(* ======================================Schrittkette======================================== *)
fb_state_entry(
	i16_next_step:= ,
	i16_pos:= 1,
	s_debugtext:= ,
	E=> ,
	X=> ,
	i16_step=> ,
	i16_last_step=> );

CASE fb_state_entry.i16_step OF
(*=======================================================*)
	INIT_OBJ:
		IF st_config_achse.b_config_fertig THEN
			fb_state_entry.i16_next_step := 2;
		END_IF

(*=======================================================*)
	2:	(* Antriebsbegrenzende Konstantwerte *)
		IF fb_state_entry.E THEN
			CASE gst_datensatz.st_md.i16_typ_zelle OF
				KEINE_ZELLE:
					;

				BESTUECKZELLE_1700 :
					st_geschwindigkeiten.lr_auto_max := 350;	(* Hub/min *)
					st_geschwindigkeiten.lr_auto_min := 15;
					st_geschwindigkeiten.lr_jog := 50;
					gst_datensatz.st_md.st_md_bestueckachse.lr_startposition := 17;

				BESTUECKZELLE_1720:
					st_geschwindigkeiten.lr_auto_max := 300;	(* Hub/min *)
					st_geschwindigkeiten.lr_auto_min := 15;
					st_geschwindigkeiten.lr_jog := 50;
					gst_datensatz.st_md.st_md_bestueckachse.lr_startposition := 3;

				RASTERFOLIE:
					st_geschwindigkeiten.lr_auto_max := 300;	(* Hub/min *)
					st_geschwindigkeiten.lr_auto_min := 15;
					st_geschwindigkeiten.lr_jog := 50;
					gst_datensatz.st_md.st_md_bestueckachse.lr_startposition := 17;
			END_CASE

			fb_state_entry.i16_next_step := 3;
		END_IF

(*=======================================================*)
	3:	(* Spezifische NC-Achsparameter auslesen *)
		IF fb_state_entry.E THEN
			subr_ST_Bandeinzugsnocken_ein();
			fb_virt_master_axis.i16_nc_parameter_nummer := MaxVelocitySystem;
			st_drive_cmd.enu_cmd := READ_NC_PARAMETER;
		END_IF

		(*-----------------------Weiterschaltbedingungen----------------------------*)
		IF st_drive_cmd.enu_cmd = NO_COMMAND THEN
			st_geschwindigkeiten.lr_maximalgeschwindigkeit := fb_virt_master_axis.r_wert_nc_read_parameter(* °/s *) * 60 / 360;
			fb_state_entry.i16_next_step := 4;
		END_IF

(*=======================================================*)
	4:	(* Spezifische NC-Achsparameter auslesen *)
		IF fb_state_entry.E THEN
			fb_virt_master_axis.i16_nc_parameter_nummer := MaxAccelerationSystem;
			st_drive_cmd.enu_cmd := READ_NC_PARAMETER;
		END_IF

		(*-----------------------Weiterschaltbedingungen----------------------------*)
		IF st_drive_cmd.enu_cmd = NO_COMMAND THEN
			st_geschwindigkeiten.lr_beschleunigung := fb_virt_master_axis.r_wert_nc_read_parameter;
			fb_state_entry.i16_next_step := 5;
		END_IF

(*=======================================================*)
	5:	(* Spezifische NC-Achsparameter auslesen *)
		IF fb_state_entry.E THEN
			fb_virt_master_axis.i16_nc_parameter_nummer := MaxDecelerationSystem;
			st_drive_cmd.enu_cmd := READ_NC_PARAMETER;
		END_IF

		(*-----------------------Weiterschaltbedingungen----------------------------*)
		IF st_drive_cmd.enu_cmd = NO_COMMAND THEN
			st_geschwindigkeiten.lr_verzoegerung := fb_virt_master_axis.r_wert_nc_read_parameter;
			lr_decceleration_normal := st_geschwindigkeiten.lr_verzoegerung;
			lr_decceleration_nothalt := 200000.0;
			fb_state_entry.i16_next_step := 6;
		END_IF

(*=======================================================*)
	6:	(* Spezifische NC-Achsparameter auslesen *)
		IF fb_state_entry.E THEN
			fb_virt_master_axis.i16_nc_parameter_nummer := MaxJerk;
			st_drive_cmd.enu_cmd := READ_NC_PARAMETER;
		END_IF

		(*-----------------------Weiterschaltbedingungen----------------------------*)
		IF st_drive_cmd.enu_cmd = NO_COMMAND THEN
			st_geschwindigkeiten.lr_ruck := fb_virt_master_axis.r_wert_nc_read_parameter;
		fb_state_entry.i16_next_step := FEHLER; (*in Fehler gehen damit die Achsen resetet werden. Sonst steigen die Achsen bei einem TC Restart aus*)
		END_IF

(*=======================================================*)
	INIT:
		IF fb_state_entry.E THEN
			fb_ton_wz.IN := FALSE;
			fb_ton_uez.IN	:= FALSE;
			fb_ton_quitt.IN := FALSE;
			fb_ton_wz_disable.IN := FALSE;
			st_ctrl_out.b_fehler := FALSE;
			st_ctrl_out.b_fertig := FALSE;
			st_ctrl_out.b_bereit := FALSE;
			st_ctrl_out.b_prebereit := FALSE;
			b_merker_bandende_links := FALSE;
			b_merker_bandende_rechts := FALSE;

			(* Reset Stoermeldungen *)
			st_sm.b_achse_nicht_auf_startpos := FALSE;
			st_sm.b_achsfehler := FALSE;
			st_sm.b_devicefehler := FALSE;
			st_sm.b_keine_verfahrfreigabe := FALSE;
			st_sm.b_ende_skalierungs_nocke := FALSE;
			st_sm.b_ende_camming_nocke := FALSE;
			st_sm.b_skalierung_noch_aktiv := FALSE;
			sm_fehler_bestueckanzahl := FALSE;
			sm_fehler_bestueckposition_z := FALSE;
			sm_fehler_positionierung_z := FALSE;
			sm_fehler_bestueckposition_y := FALSE;
			sm_fehler_positionierung_y := FALSE;
			sm_fehler_achse_lueften := FALSE;
			sm_fehler_raster_oder_zaehne := FALSE;
			sm_fehler_bestueckschieberanzahl := FALSE;
			sm_keine_busverbindung := FALSE;
			sm_fehler_nach_bandwechsel := FALSE;
			sm_fehler_positionierung_bestueckachse := FALSE;

			(* Reset Betriebsmeldungen *)
			bm_bandende_einzug_links_erreicht := FALSE;
			bm_bandende_einzug_rechts_erreicht := FALSE;
			bm_bandende_beide_einzuege_erreicht := FALSE;
			bm_einzug_links_band_entnehmen := FALSE;
			bm_einzug_links_band_auf_anschlag := FALSE;
			bm_einzug_rechts_band_entnehmen := FALSE;
			bm_einzug_rechts_band_auf_anschlag := FALSE;
			bm_einzug_rechts_band_bis_gls := FALSE;
			bm_einzug_links_band_bis_gls := FALSE;
			bm_beide_Bandklemmen_oeffnen := FALSE;
			bm_an_visu_hinten := '';

			ST_TippTasten.b_einfaedeln_aktiv := FALSE;
			bandwechsel_kontroller.st_ctrl.in.b_start := FALSE;
			einpresskraft_kontroller.st_ctrl.in.b_start := FALSE;
			bandeinzug_kontroller.st_ctrl.in.b_freigabe := FALSE;
			axis_bandeinzug_achse.st_ctrl.in.b_freigabe := FALSE;
			axis_bandeinzug_achse.st_ctrl.in.b_bremse_auf := FALSE;
			axis_bandeinzug_achse.st_ctrl.in.b_bremse_zu := FALSE;
			axis_bandeinzug_achse.st_ctrl.in.b_start_schreiben := FALSE;
			axis_bandeinzug_achse.st_ctrl.in.b_start := FALSE;
			axis_bandeinzug_achse.st_ctrl.in.b_home := FALSE;
			axis_bandeinzug_achse.st_ctrl.in.b_ausfaedeln_servo := FALSE;
			axis_bandeinzug_achse.st_ctrl.in.b_einfaedeln_servo := FALSE;

			fb_berechnung_override_achse.lr_skalierung_slave_achse1 := 1;
			fb_berechnung_override_achse.lr_skalierung_slave_achse2 := 1;

			i16_step_lueften := 0;
			i16_einfaedelzaehler := 0;

			st_geschwindigkeiten.lr_verzoegerung := lr_decceleration_normal;

			b_bestueckschieber_ueberwachung_aktiv := TRUE;

			b_einfaedeln_aktiv_servo := FALSE;

			gb_memEndOfBandMarkNIO := FALSE;
		END_IF

		(* Gearout/Camout der Slaveachsen, damit diese quittiert werden können *)
		CASE gst_datensatz.st_md.i16_typ_zelle OF
			KEINE_ZELLE:
				;

			BESTUECKZELLE_1700:
				IF bestueckachse.NcToPlc.CoupleState > 0 THEN
					st_drive_cmd_bestueckachse.enu_cmd := CAM_OUT_SLAVE;
				END_IF
				IF z_achse.NcToPlc.CoupleState > 0 THEN
					st_drive_cmd_z_achse.enu_cmd := CAM_OUT_SLAVE;
				END_IF
				IF y_achse.NcToPlc.CoupleState > 0 THEN
					st_drive_cmd_y_achse.enu_cmd := CAM_OUT_SLAVE;
				END_IF

				CASE gst_datensatz.st_wkz.i16_typ_bandeinzug OF
					KEIN_EINZUG:
						;
					STANDARD_2FACH_V2:
						;
					 BANDWECHSLER_V2:
						;
					SERVO:
						IF b_achse.NcToPlc.CoupleState > 0 THEN
							st_drive_cmd_b_achse.enu_cmd := CAM_OUT_SLAVE;
						END_IF
				END_CASE

			BESTUECKZELLE_1720:
				IF bestueckachse.NcToPlc.CoupleState > 0 THEN
					st_drive_cmd_bestueckachse.enu_cmd := CAM_OUT_SLAVE;
				END_IF
				IF z_achse.NcToPlc.CoupleState > 0 THEN
					st_drive_cmd_z_achse.enu_cmd := CAM_OUT_SLAVE;
				END_IF

			RASTERFOLIE:
				IF bestueckachse.NcToPlc.CoupleState > 0 THEN
					st_drive_cmd_bestueckachse.enu_cmd := CAM_OUT_SLAVE;
				END_IF
				IF z_achse.NcToPlc.CoupleState > 0 THEN
					st_drive_cmd_z_achse.enu_cmd := CAM_OUT_SLAVE;
				END_IF
		END_CASE

		(*-----------------------Weiterschaltbedingungen----------------------------*)
		IF st_ctrl_in.b_preinit THEN
			fb_state_entry.i16_next_step := 12;
		END_IF

(*=======================================================*)
	12:	(* Reglerfreigabe wegnehmen *)
		IF fb_state_entry.E THEN
			st_drive_cmd.enu_cmd := POWER_DISABLE;
		END_IF

		(*-----------------------Weiterschaltbedingungen----------------------------*)
		IF st_drive_cmd.enu_cmd = NO_COMMAND THEN
			fb_state_entry.i16_next_step := 14;
		END_IF

(*=======================================================*)
	14:	(* Lade Wkz von Festplatte *)
		IF fb_state_entry.E THEN
			gi16_bbgen_auftrag := LESE_WKZ;
		END_IF

		IF  gi16_bbgen_auftrag = KEIN_BB_AUFTRAG THEN
			fb_ton_wz.pt := t#5ms;
			fb_ton_wz.IN := TRUE;
		END_IF

		IF fb_ton_wz.Q THEN
			fb_state_entry.i16_next_step := 16;
			fb_ton_wz.IN := FALSE;
		END_IF

(*=======================================================*)
	16: (* Band aus DB von Festplatte einlesen. *)
		IF fb_state_entry.E THEN
			gi16_bbgen_auftrag := LESE_BAND;
		END_IF

		IF  gi16_bbgen_auftrag = KEIN_BB_AUFTRAG THEN
			fb_ton_wz.pt := t#5ms;
			fb_ton_wz.IN := TRUE;
		END_IF

		IF fb_ton_wz.Q THEN
			fb_state_entry.i16_next_step := 20;
			fb_ton_wz.IN := FALSE;
		END_IF

(*=======================================================*)
	20:	(* CAM_OUT Bestückachse *)
		IF fb_state_entry.E THEN
			st_drive_cmd_bestueckachse.enu_cmd := CAM_OUT_SLAVE;
		END_IF

		(*-----------------------Weiterschaltbedingungen----------------------------*)
		IF st_drive_cmd_bestueckachse.enu_cmd = NO_COMMAND AND NOT fb_state_entry.E THEN
			fb_state_entry.i16_next_step := 30;
		END_IF

(*=======================================================*)
	30:	(* CAM Out Z-Achse *)
		IF fb_state_entry.E THEN
			st_drive_cmd_z_achse.enu_cmd := CAM_OUT_SLAVE;
		END_IF

		(*-----------------------Weiterschaltbedingungen----------------------------*)
		IF st_drive_cmd_z_achse.enu_cmd = NO_COMMAND AND NOT fb_state_entry.E THEN
			CASE gst_datensatz.st_md.i16_typ_zelle OF
				KEINE_ZELLE:
					;

				BESTUECKZELLE_1700:
					CASE gst_datensatz.st_wkz.i16_typ_bandeinzug OF
						KEIN_EINZUG,  STANDARD_2FACH_V2,  BANDWECHSLER_V2:
							fb_state_entry.i16_next_step := 40;
						SERVO:
							fb_state_entry.i16_next_step := 35;
					END_CASE;

				RASTERFOLIE:
					fb_state_entry.i16_next_step := 40;

				BESTUECKZELLE_1720:
					fb_state_entry.i16_next_step := 45;
			END_CASE
		END_IF

(*=======================================================*)
	35:	(* CAM Out B-Achse *)
		IF fb_state_entry.E THEN
			st_drive_cmd_b_achse.enu_cmd := CAM_OUT_SLAVE;
		END_IF

		(*-----------------------Weiterschaltbedingungen----------------------------*)
		IF st_drive_cmd_b_achse.enu_cmd = NO_COMMAND AND NOT fb_state_entry.E THEN
			fb_state_entry.i16_next_step := 40;
		END_IF

(*=======================================================*)
	40:	(* CAM Out Y-Achse *)
		IF fb_state_entry.E THEN
			st_drive_cmd_y_achse.enu_cmd := CAM_OUT_SLAVE;
		END_IF

		(*-----------------------Weiterschaltbedingungen----------------------------*)
		IF st_drive_cmd_y_achse.enu_cmd = NO_COMMAND AND NOT fb_state_entry.E THEN
			fb_state_entry.i16_next_step := 45;
		END_IF

(*=======================================================*)
	45:	(* Reglerfreigabe setzen , Reset wird bei Bedarf automatisch ausgeführt*)
		IF fb_state_entry.E THEN
			st_drive_cmd.enu_cmd := POWER_ENABLE;
		END_IF

		(*-----------------------Weiterschaltbedingungen----------------------------*)
		IF st_drive_cmd.enu_cmd = NO_COMMAND THEN
			fb_state_entry.i16_next_step := 50;
		END_IF

(*=======================================================*)
	50:
		IF fb_state_entry.E THEN
			st_ctrl_out.b_prebereit := TRUE;
		END_IF

		(*-----------------------Weiterschaltbedingungen----------------------------*)
		IF st_ctrl_in.b_init THEN
			fb_state_entry.i16_next_step := 60;
		END_IF

(*=======================================================*)
	60:  (* Die Masterachsposition auf Startposition der Bestückachse setzen *)
		CASE gst_datensatz.st_md.i16_typ_zelle OF
			KEINE_ZELLE:
				;

			BESTUECKZELLE_1700, BESTUECKZELLE_1720, RASTERFOLIE:
				IF fb_state_entry.E THEN
					fb_virt_master_axis.st_position.r_soll := gst_datensatz.st_md.st_md_bestueckachse.lr_startposition;
					st_drive_cmd.enu_cmd := SET_POSITION;
				END_IF
		END_CASE

		(*-----------------------Weiterschaltbedingungen----------------------------*)
		IF st_drive_cmd.enu_cmd = NO_COMMAND THEN
			fb_state_entry.i16_next_step := 70;
		END_IF

(*=======================================================*)
	70:	(* Camin Bestückachse -> synchronisiere sofort Virtuelle Masterachse mit Bestückachse *)
		IF fb_state_entry.E THEN
			i16_bestueckachse_cam_table_id := 5;
			fb_axis_bestueckachse.st_camscaling_data.SlaveScaling := axis_bestueckachse.st_config.r_getriebefaktor;
			fb_axis_bestueckachse.mc_activation_mode_camin:= MC_CAMACTIVATION_INSTANTANEOUS;
			fb_axis_bestueckachse.lr_activation_position_camin := gst_datensatz.st_md.st_md_bestueckachse.lr_startposition;
			st_drive_cmd_bestueckachse.enu_cmd := CAM_IN_SLAVE;
			i16_bestueckachse_cam_table_id_alt := i16_bestueckachse_cam_table_id;
		END_IF

		(*-----------------------Weiterschaltbedingungen----------------------------*)
		IF st_drive_cmd_bestueckachse.enu_cmd = NO_COMMAND AND NOT fb_state_entry.E THEN
			fb_state_entry.i16_next_step := 80;
		END_IF

(*=======================================================*)
	80: (* Prüfe Bandeinzugsdaten wenn Servo verwendet wird => Verhindere Div by 0 *)
		IF fb_state_entry.E THEN
			IF gst_datensatz.st_wkz.i16_typ_bandeinzug = SERVO THEN
				IF gst_datensatz.st_band.r_raster < 0.05 OR
					gst_datensatz.st_band.i16_igelrad_zaehne <= 0 THEN
					sm_fehler_raster_oder_zaehne := TRUE;
					fb_state_entry.i16_next_step := FEHLER;;
				END_IF
			END_IF
		END_IF

		(*-----------------------Weiterschaltbedingungen----------------------------*)
		IF fb_state_entry.i16_next_step <> FEHLER AND NOT fb_state_entry.E THEN
			fb_state_entry.i16_next_step := BEREIT;
		END_IF

(*=======================================================*)
	BEREIT:
		IF fb_state_entry.E THEN
			st_ctrl_out.b_bereit := TRUE;
			st_ctrl_out.b_fertig := TRUE;
			i16_bestueckposzaehler := 0;
			bandeinzug_kontroller.st_ctrl.in.b_freigabe := FALSE;
			axis_bandeinzug_achse.st_ctrl.in.b_freigabe := FALSE;
		END_IF

		(* Bedienergeführter Einfädelablauf mit Anstanzprogramm aus der Grundstellung. *)
		CASE gst_datensatz.st_md.i16_typ_zelle OF
			KEINE_ZELLE:
				;

			BESTUECKZELLE_1700:
				CASE gst_datensatz.st_wkz.i16_typ_bandeinzug OF
					 BANDWECHSLER_V2:
						IF NOT gst_datensatz.st_md.b_wt_transport_simulation THEN
							IF NOT fb_tof_bandende_li.Q AND zyl_bawe_querschub.fb.e_sensor1_eingefahren THEN
								bm_bandende_einzug_links_erreicht := TRUE;
								b_merker_bandende_links := TRUE;
								i16_merker_last_state := fb_state_entry.i16_step;
								fb_state_entry.i16_next_step :=300;	(* ->Bandwechsel *)
							ELSIF NOT fb_tof_bandende_re.Q AND zyl_bawe_querschub.fb.e_sensor1_ausgefahren THEN
								bm_bandende_einzug_rechts_erreicht := TRUE;
								b_merker_bandende_rechts := TRUE;
								i16_merker_last_state := fb_state_entry.i16_step;
								fb_state_entry.i16_next_step := 300;	(* ->Bandwechsel *)
							END_IF
						END_IF

					SERVO:
						IF NOT gst_datensatz.st_md.b_wt_transport_simulation THEN
							IF NOT fb_tof_bandende_li.Q AND zyl_bawe_querschub.fb.e_sensor1_eingefahren THEN
								bm_bandende_einzug_links_erreicht := TRUE;
								b_merker_bandende_links := TRUE;
								i16_merker_last_state := fb_state_entry.i16_step;
								fb_state_entry.i16_next_step := 640;
							ELSIF  NOT fb_tof_bandende_re.Q AND zyl_bawe_querschub.fb.e_sensor1_ausgefahren THEN
								bm_bandende_einzug_rechts_erreicht := TRUE;
								b_merker_bandende_rechts := TRUE;
								i16_merker_last_state := fb_state_entry.i16_step;
								fb_state_entry.i16_next_step := 640;
							END_IF
						END_IF
				END_CASE;


			BESTUECKZELLE_1720:
				CASE gst_datensatz.st_wkz.i16_typ_bandeinzug OF
					  STANDARD_2FACH_V2:
						IF NOT gst_datensatz.st_md.b_wt_transport_simulation THEN
							(* Band wird nur am Steckeranfang nach Neueinfädeln angestanzt. *)
							IF NOT fb_tof_bandende_li.Q OR NOT fb_tof_bandende_re.Q THEN
								b_merker_bandende_links := TRUE;
								b_merker_bandende_rechts := TRUE;
								bm_bandende_beide_einzuege_erreicht := TRUE;
								i16_merker_last_state := fb_state_entry.i16_step;
								fb_state_entry.i16_next_step := 420;
							END_IF
						END_IF
				END_CASE

			RASTERFOLIE:
				(*Beim 92 pol. Stecker muss eine Einfädelroutine gestartet werden*)
				IF gst_datensatz.st_wkz.b_rafo_auto_einf_aktiv AND NOT fb_tof_bandende_rafo.Q THEN
					bm_bandende_einzug_links_erreicht := TRUE;
					fb_state_entry.i16_next_step := 810;
				END_IF
		END_CASE

		(*-----------------------Weiterschaltbedingungen----------------------------*)
		IF fb_r_trig_start.Q AND NOT fb_state_entry.E THEN
			st_ctrl_out.b_fertig := FALSE;
			ST_TippTasten.b_einfaedeln_aktiv := FALSE;
			b_einfaedeln_aktiv_servo := FALSE;
			bandeinzug_kontroller.st_ctrl.in.b_freigabe := TRUE;
			gb_memEndOfBandMarkNIO := FALSE;
			fb_state_entry.i16_next_step := 110;
			IF gst_barcode_daten.b_band_links_ok THEN
				b_merker_bandende_links := FALSE;
			END_IF
			IF gst_barcode_daten.b_band_rechts_ok THEN
				b_merker_bandende_rechts := FALSE;
			END_IF
		ELSIF fb_r_trig_start_remove_pos.Q AND NOT fb_state_entry.E THEN
			fb_state_entry.i16_next_step := 900;
		END_IF

(*=======================================================*)
	110:	(* Auswahl als was die Zelle Betrieben wird *)
		IF fb_state_entry.E THEN
			CASE gst_datensatz.st_md.i16_typ_zelle OF
				KEINE_ZELLE:
					;

				BESTUECKZELLE_1700, BESTUECKZELLE_1720:
					fb_state_entry.i16_next_step := 130;

				RASTERFOLIE:
					fb_state_entry.i16_next_step := 800;
			END_CASE
		END_IF

(*=========================Regulärer Bestückablauf==============================*)
	130:	(* Fahre vorgegebene Anzahl von Bestückhüben *)
		IF fb_state_entry.E THEN
			fb_virt_master_axis.st_position.r_soll := (DINT_TO_LREAL(gst_datensatz.st_bestueckprogramm.i32_anzahl)) * 360.0 + gst_datensatz.st_md.st_md_bestueckachse.lr_startposition;
			st_drive_cmd.enu_cmd := MOVE_MODULO;	(* Achtung beim MODULO-Befehl: fährt nur bis 360° *)
			fb_virt_master_axis.mc_richtung_modulo :=MC_Positive_Direction ;
		END_IF

		(*-----------------------Weiterschaltbedingungen----------------------------*)
		fb_state_entry.i16_next_step := 140;

(*=======================================================*)
	140:	(* Positionsmerker für die Bestückpositionsüberwachung *)
		IF fb_state_entry.E THEN
			lr_merker_z_pos := gst_datensatz.st_isk.lr_pos_z_0 + gst_datensatz.st_wkz.lr_offset_z_pos_0 + gst_datensatz.st_wt.lr_offset_z_pos_0 + gst_datensatz.st_md.lr_offset_z_pos_0;
			lr_merker_y_pos := gst_datensatz.st_isk.lr_pos_y_0 + gst_datensatz.st_wkz.lr_offset_y_pos_0 + gst_datensatz.st_wt.lr_offset_y_pos_0 + gst_datensatz.st_md.lr_offset_y_pos_0;
			subr_ST_Cam_Bestueck_Maschine();
		END_IF

		(*-----------------------Weiterschaltbedingungen----------------------------*)
		fb_state_entry.i16_next_step := 150;

(*=======================================================*)
	150:	(* Bestückachse läuft im Getriebegleichlauf, die Z-Achse bzw. Y-Achse wird gekoppelt oder skaliert *)
		IF fb_state_entry.E THEN
			lr_merker_z_pos_alt := 500.0;	(* einfach ein Wert ausserhalb des Verfahrbereichs der Z-Achse *)
			lr_merker_y_pos_alt := 100.0;	(* einfach ein Wert ausserhalb des Verfahrbereichs der Y-Achse *)

			einpresskraft_kontroller.st_ctrl.in.b_start := TRUE;

			IF gst_datensatz.st_wkz.i16_typ_bandeinzug = SERVO THEN
				axis_bandeinzug_achse.st_ctrl.in.b_freigabe := TRUE;
			END_IF
		END_IF

		IF gst_datensatz.st_md.i16_typ_zelle = BESTUECKZELLE_1700 THEN
			(*Überwachungsfunktion, ob das Auskoppeln der Bestückachse geklappt hat.*)
			subr_ST_PosUW_Bestueckachse();
		END_IF

		IF fb_r_trig_bestueckhubzaehler.Q THEN
			CASE gst_datensatz.st_md.i16_typ_zelle OF
				KEINE_ZELLE:
					;
				BESTUECKZELLE_1700:
					(* Positionsüberwachung Achsen *)
					CASE gst_datensatz.st_wkz.i16_typ_bandeinzug OF
						 BANDWECHSLER_V2:
							subr_ST_PosUW_YZ_Achse();

						SERVO:
							subr_ST_PosUW_YZ_Achse();
							subr_ST_B_Achse();
					END_CASE;
					(* Zählt die gesetzten Pins während des gesamten Bestückvorganges *)
					i16_bestueckposzaehler := i16_bestueckposzaehler + 1;

					(* >>>>>>>>>>>>>>>>>>>><<<<<<<<<<<<<<<<<<< *)
					(*
					Diese Änderung wurde 1:1 aus Tschechien übernommen.
					Merker "gb_memEndOfBandMarkNIO" für Bandende während des Bestückens. Diese Variable gilt nur
					für den One27 in Tschechien. Während des Bestückens wird der Bandende Sensor abgefragt. Wenn
					noch mehr wie 80 Pins zu bestücken sind und der Bandende Sensor anschlägt, wird ein "HALT_AXIS"
					der virtuellen Masterachse ausgeführt. Die Achse bleibt zufällig irgendwo stehen. Der WT bleibt auf
					Bestückposition stehen. Eine Fehlermeldung kommt vom Bandwechselkontroller. Dann muss die 
					Anlage quittiert werden. Bestückachse fährt in Grundstellung und WT fährt auf Übergabeposition.
					Danach wird der Bandwechselvorgang gestartet. *)
					i16_LeftPins := DINT_TO_INT(gst_datensatz.st_bestueckprogramm.i32_anzahl) - i16_bestueckposzaehler;
					IF (NOT fb_tof_bandende_li.Q) AND
						(F_ToUCase(gst_bestueckbild_halbauto.s_beschreibung) = 'ONE27') AND
						(i16_LeftPins > 80) THEN
						i16_bestueckposzaehler := DINT_TO_INT(gst_datensatz.st_bestueckprogramm.i32_anzahl);
						gb_memEndOfBandMarkNIO := TRUE;
						st_drive_cmd.enu_cmd := HALT_AXIS;
					END_IF
					(* >>>>>>>>>>>>>>>>>>>><<<<<<<<<<<<<<<<<<< *)

				BESTUECKZELLE_1720:
					(* Positionsüberwachung Achsen *)
					CASE gst_datensatz.st_wkz.i16_typ_bandeinzug OF
						STANDARD_2FACH_V2:
							subr_ST_PosUW_Z_Achse();
						SERVO:
							subr_ST_B_Achse();
					END_CASE;
					(* Zählt die gesetzten Pins während des gesamten Bestückvorganges *)
					i16_bestueckposzaehler := i16_bestueckposzaehler + 1;

				RASTERFOLIE:
					;
			END_CASE
		END_IF

		(* Auf Startposition achten, damit die Erstskalierung nicht übersehen wird *)
		IF i16_bestueckposzaehler >= 0 AND i16_bestueckposzaehler <= gst_datensatz.st_bestueckprogramm.i32_anzahl THEN
			(* Warte auf OT-Nocken für Skalierungsfreigabe *)
			IF fb_f_trig_ot.Q THEN
				subr_ST_Cam_Bestueck_Maschine();
			END_IF

			(* Warte auf Nocken für die Skalierungsfreigabe *)
			IF fb_r_trig_skalierungsnocken.Q THEN
				CASE gst_datensatz.st_md.i16_typ_zelle OF
					KEINE_ZELLE:
						;
					BESTUECKZELLE_1700:
						CASE gst_datensatz.st_wkz.i16_typ_bandeinzug OF
							 BANDWECHSLER_V2:
								(* Skalierung der Kurvenscheibe *)
								subr_ST_Cam_Z_Achse();
								subr_ST_Cam_Y_Achse();

							SERVO:
								(* Skalierung der Kurvenscheibe *)
								subr_ST_Cam_Z_Achse();
								subr_ST_Cam_Y_Achse();
								subr_ST_Cam_B_Achse();
						END_CASE;

					BESTUECKZELLE_1720:
						CASE gst_datensatz.st_wkz.i16_typ_bandeinzug OF
							STANDARD_2FACH_V2:
								(* Skalierung der Kurvenscheibe *)
								subr_ST_Cam_Z_Achse();
						END_CASE;

					RASTERFOLIE:
						;
				END_CASE
			END_IF
		END_IF

		(*====================================================================================================================*)
		IF  i16_bestueckposzaehler = gst_datensatz.st_bestueckprogramm.i32_anzahl THEN
			(* Wenn alle Bestückhübe gemacht sind warte auf Bestückachse im Ziel *)
			CASE gst_datensatz.st_md.i16_typ_zelle OF
				KEINE_ZELLE:
					;
				BESTUECKZELLE_1700:
					CASE gst_datensatz.st_wkz.i16_typ_bandeinzug OF
						 BANDWECHSLER_V2:
							IF	virtuelle_master_achse.Status.NotMoving  AND
								virtuelle_master_achse.Status.InTargetPosition AND
								st_drive_cmd.enu_cmd = NO_COMMAND 	AND
								st_drive_cmd_z_achse.enu_cmd = NO_COMMAND AND
								st_drive_cmd_y_achse.enu_cmd = NO_COMMAND
								THEN
									(* Kontrolle, ob die gemachten Bestückhübe der Vorgabe aus dem Bestückprogramm entsprechen *)
									IF i16_bestueckposzaehler = gst_datensatz.st_bestueckprogramm.i32_anzahl THEN
										fb_state_entry.i16_next_step := 170;
									ELSE
										sm_fehler_bestueckanzahl := TRUE;
										fb_state_entry.i16_next_step := FEHLER;
									END_IF
							END_IF

						SERVO:
							IF	virtuelle_master_achse.Status.NotMoving  AND
								virtuelle_master_achse.Status.InTargetPosition AND
								st_drive_cmd.enu_cmd = NO_COMMAND 	AND
								st_drive_cmd_z_achse.enu_cmd = NO_COMMAND AND
								st_drive_cmd_y_achse.enu_cmd = NO_COMMAND AND
								st_drive_cmd_b_achse.enu_cmd = NO_COMMAND
								THEN
									(* Kontrolle, ob die gemachten Bestückhübe der Vorgabe aus dem Bestückprogramm entsprechen *)
									IF i16_bestueckposzaehler = gst_datensatz.st_bestueckprogramm.i32_anzahl THEN
										fb_state_entry.i16_next_step := 160;
									ELSE
										sm_fehler_bestueckanzahl := TRUE;
										fb_state_entry.i16_next_step := FEHLER;
									END_IF
							END_IF
					END_CASE;

				BESTUECKZELLE_1720:
					CASE gst_datensatz.st_wkz.i16_typ_bandeinzug OF
						 STANDARD_2FACH_V2:
							IF	virtuelle_master_achse.Status.NotMoving  AND
								virtuelle_master_achse.Status.InTargetPosition AND
								st_drive_cmd.enu_cmd = NO_COMMAND 	AND
								st_drive_cmd_z_achse.enu_cmd = NO_COMMAND
								THEN
									(* Kontrolle, ob die gemachten Bestückhübe der Vorgabe aus dem Bestückprogramm entsprechen *)
									IF i16_bestueckposzaehler = gst_datensatz.st_bestueckprogramm.i32_anzahl THEN
										fb_state_entry.i16_next_step := 180;
									ELSE
										sm_fehler_bestueckanzahl := TRUE;
										fb_state_entry.i16_next_step := FEHLER;
									END_IF
							END_IF
					END_CASE

				RASTERFOLIE:
					;
			END_CASE
		END_IF

		(* Nach dem ersten WT wird die Bestückschieberüberwachung ausgeschaltet (Wunsch von Häußerer Josy) *)
		(* Bei der Grundstellungsfahrt wird die Abfrage wieder aktiviert *)
		IF fb_state_entry.X THEN
			axis_bandeinzug_achse.st_ctrl.in.b_freigabe := FALSE;
			gst_datensatz.st_wkz.nockenschaltwerk_bestueckachse.arr_nocken[NO_UW_BESTUECKSCHIEBER_ON].b_camvalid := FALSE;
			gst_datensatz.st_wkz.nockenschaltwerk_bestueckachse.arr_nocken[NO_UW_BESTUECKSCHIEBER_OFF].b_camvalid := FALSE;
			gst_datensatz.st_wkz.nockenschaltwerk_bestueckachse.arr_nocken[SP_UW_BESTUECKSCHIEBER_ON].b_camvalid := FALSE;
			gst_datensatz.st_wkz.nockenschaltwerk_bestueckachse.arr_nocken[SP_UW_BESTUECKSCHIEBER_OFF].b_camvalid := FALSE;
			b_bestueckschieber_ueberwachung_aktiv := FALSE;
			einpresskraft_kontroller.st_ctrl.in.b_start := FALSE;
		END_IF

(*=======================================================*)
	160:	(* Kopplung mit B-Achse lösen *)
		IF fb_state_entry.E THEN
			st_drive_cmd_b_achse.enu_cmd := CAM_OUT_SLAVE;
		END_IF

		(*-----------------------Weiterschaltbedingungen----------------------------*)
		IF st_drive_cmd_b_achse.enu_cmd = NO_COMMAND THEN
			fb_state_entry.i16_next_step := 170;
		END_IF

(*=======================================================*)
	170:	(* Kopplung mit Y-Achse lösen *)
		IF fb_state_entry.E THEN
			fb_berechnung_override_achse.lr_skalierung_slave_achse2 := 1;
			st_drive_cmd_y_achse.enu_cmd := CAM_OUT_SLAVE;
		END_IF

		(*-----------------------Weiterschaltbedingungen----------------------------*)
		IF st_drive_cmd_y_achse.enu_cmd = NO_COMMAND THEN
			fb_state_entry.i16_next_step := 180;
		END_IF

(*=======================================================*)
	180:	(* Kopplung mit Z-Achse lösen *)
		IF fb_state_entry.E THEN
			fb_berechnung_override_achse.lr_skalierung_slave_achse1 := 1;
			st_drive_cmd_z_achse.enu_cmd := CAM_OUT_SLAVE;
		END_IF

		(*-----------------------Weiterschaltbedingungen----------------------------*)
		IF st_drive_cmd_z_achse.enu_cmd = NO_COMMAND THEN
			fb_state_entry.i16_next_step := BEREIT;
		END_IF

(*=======================================================*)
	300:	(* Cam_in_Slave*)
		IF fb_state_entry.E THEN
			subr_ST_Bandeinzugsnocken_aus();
			bandeinzug_kontroller.st_ctrl.in.b_freigabe := FALSE;           (* GLS überwachung ausschalten*)
			ST_TippTasten.b_einfaedeln_aktiv := TRUE;
			i16_bestueckachse_cam_table_id := 5;
			fb_axis_bestueckachse.mc_activation_mode_camin:= MC_CAMACTIVATION_ATMASTERCAMPOS;
			fb_axis_bestueckachse.lr_activation_position_camin := gst_datensatz.st_md.st_md_bestueckachse.lr_startposition;
			st_drive_cmd_bestueckachse.enu_cmd := CAM_IN_SLAVE;
			i16_bestueckachse_cam_table_id_alt := i16_bestueckachse_cam_table_id;
		END_IF

		(*-----------------------Weiterschaltbedingungen----------------------------*)
		IF st_drive_cmd_bestueckachse.enu_cmd = NO_COMMAND AND NOT fb_state_entry.E THEN
			fb_state_entry.i16_next_step :=305;
		END_IF

(*===========================Anstanzen 1700 mit Klemmbandeinzug V2============================*)
	305:	(* Nocken sind deaktiviert, Bandeinzug ist bereits ausgeschaltet, jetzt beide Zylinder lösen. *)
		IF fb_state_entry.E THEN
			(* Band freigeben für Bedienerentnahme *)
			bandwechsel_kontroller.st_ctrl.in.b_start := TRUE;
			zyl_bandfaenger.st_ctrl.in.b_einfahren := TRUE;
			zyl_bandklemmen.st_ctrl.in.b_einfahren := TRUE;
			gi16_anzahl_Teile_autostop_bandwechsel := 0;
		END_IF

		(*-----------------------Weiterschaltbedingungen----------------------------*)
		IF NOT bandwechsel_kontroller.st_ctrl.out.b_fertig AND NOT bandwechsel_kontroller.st_ctrl.out.b_fertig_2 THEN
			fb_state_entry.i16_next_step := 306;
		END_IF

(*=======================================================*)
	306:	(* Warten auf Bandwechselkontroller fertig*)

		(*-----------------------Weiterschaltbedingungen----------------------------*)
		(*Einfädeln nach automatischem Bandwechsel*)
		IF bandwechsel_kontroller.st_ctrl.out.b_fertig AND NOT fb_state_entry.E THEN
			bandwechsel_kontroller.st_ctrl.in.b_start := FALSE;
			bm_bandende_einzug_links_erreicht := FALSE;
			bm_bandende_einzug_rechts_erreicht := FALSE;
			b_automatischer_bandwechsel := TRUE;
			fb_state_entry.i16_next_step := 360;
		(*Einfädeln nach manuellem Bandwechsel*)
		ELSIF bandwechsel_kontroller.st_ctrl.out.b_fertig_2 AND NOT fb_state_entry.E THEN
			bandwechsel_kontroller.st_ctrl.in.b_start := FALSE;
			bm_bandende_einzug_links_erreicht := FALSE;
			bm_bandende_einzug_rechts_erreicht := FALSE;
			b_automatischer_bandwechsel := FALSE;
			fb_state_entry.i16_next_step := 310;
		END_IF

(*=======================================================*)
	310:	(* Bandende im linken oder rechten Einzug ohne Bandwechsel ->Meldung und warte auf Bediener *)
		IF fb_state_entry.E THEN
			bm_bandende_einzug_links_erreicht := FALSE;
			bm_bandende_einzug_rechts_erreicht := FALSE;
			IF b_merker_bandende_links THEN
				bm_einzug_links_band_entnehmen := TRUE;
			ELSIF b_merker_bandende_rechts THEN
				bm_einzug_rechts_band_entnehmen := TRUE;
			END_IF
			bm_an_visu_hinten :=  visu_hinten.in.texte.txt_bm_einfaedeln[0];(*Band am Einzug entnehmen -> Taste TIPPEN.*)
		END_IF

		(*-----------------------Weiterschaltbedingungen----------------------------*)
		IF ST_TippTasten.r_trig_tippen_einfaedeln.Q THEN
			(* Bei Tastendruck darf sich kein Band im Einzug befinden *)
			IF b_merker_bandende_links THEN
				IF NOT e_ls_bandende_li THEN
					fb_state_entry.i16_next_step :=320;
				END_IF
			ELSIF b_merker_bandende_rechts THEN
				IF NOT e_ls_bandende_re THEN
					fb_state_entry.i16_next_step := 320;
				END_IF
			END_IF
		ELSIF fb_r_trig_start_remove_pos.Q AND NOT fb_state_entry.E THEN
			fb_state_entry.i16_next_step := 900;
		END_IF

(*=======================================================*)
	320:	(* Fahre auf UT, Bestückachse ist wieder gekoppelt *)
		IF fb_state_entry.E THEN
			bm_einzug_links_band_entnehmen := FALSE;
			bm_einzug_rechts_band_entnehmen := FALSE;
			bm_an_visu_hinten := '';

			fb_virt_master_axis.mc_richtung_modulo :=  MC_Positive_Direction  ;
			fb_virt_master_axis.st_position.r_soll := gst_datensatz.st_wkz.lr_einfaedelposition;
			st_drive_cmd.enu_cmd := MOVE_MODULO;
		END_IF

		(*-----------------------Weiterschaltbedingungen----------------------------*)
		IF st_drive_cmd.enu_cmd = NO_COMMAND THEN
			fb_state_entry.i16_next_step := 330;
		END_IF

(*=======================================================*)
	330:	(* Meldung und warte auf Bediener *)
		IF fb_state_entry.E THEN
			IF b_merker_bandende_links THEN
				bm_einzug_links_band_auf_anschlag := TRUE;
				bm_an_visu_hinten :=  visu_hinten.in.texte.txt_bm_einfaedeln[8];(*Band an Einzug links auf Anschlag in WKZ -> Taste TIPPEN.*)
			ELSIF b_merker_bandende_rechts THEN
				bm_einzug_rechts_band_auf_anschlag := TRUE;
				bm_an_visu_hinten :=  visu_hinten.in.texte.txt_bm_einfaedeln[9];(*Band an Einzug rechts auf Anschlag in WKZ -> Taste TIPPEN*)
			END_IF
		END_IF

		IF ST_TippTasten.r_trig_tippen_einfaedeln.Q  THEN
			bm_einzug_links_band_auf_anschlag := FALSE;
			bm_einzug_rechts_band_auf_anschlag := FALSE;
			bm_an_visu_hinten := '';

			(* Klemme das Band *)
			zyl_bandklemmen.st_ctrl.in.b_einfahren := FALSE;
			zyl_bandklemmen.st_ctrl.in.b_ausfahren := TRUE;
			zyl_bandfaenger.st_ctrl.in.b_einfahren := TRUE;
			zyl_bandfaenger.st_ctrl.in.b_ausfahren := FALSE;
		END_IF

		(*-----------------------Weiterschaltbedingungen----------------------------*)
		IF zyl_bandfaenger.st_ctrl.out.b_eingefahren AND zyl_bandklemmen.st_ctrl.out.b_ausgefahren THEN
			fb_state_entry.i16_next_step := 340;
		END_IF

(*=======================================================*)
	340:	(* Warte kurz auf Zylinder *)
		IF fb_state_entry.E THEN
 			fb_ton_wz.PT := t#1s;
			fb_ton_wz.IN := TRUE;
		END_IF

		(*-----------------------Weiterschaltbedingungen----------------------------*)
		IF fb_ton_wz.Q THEN
			fb_ton_wz.IN := FALSE;
			fb_state_entry.i16_next_step := 350;
		END_IF

(*=======================================================*)
	350:	(* Fahre auf OT - Band ist geklemmt *)
		IF fb_state_entry.E THEN
			fb_virt_master_axis.mc_richtung_modulo :=  MC_Positive_Direction  ;
			fb_virt_master_axis.st_position.r_soll := gst_datensatz.st_md.st_md_bestueckachse.lr_startposition;
			st_drive_cmd.enu_cmd := MOVE_MODULO;
			bm_an_visu_hinten :=  visu_hinten.in.texte.txt_bm_einfaedeln[1];(*Werkzeug fährt auf OT.*)
		END_IF

		(*-----------------------Weiterschaltbedingungen----------------------------*)
		IF st_drive_cmd.enu_cmd = NO_COMMAND THEN
			fb_state_entry.i16_next_step := 360;
		END_IF

(*=======================================================*)
	360:	(* Die Zylinder wieder den Nocken überlassen *)
		IF fb_state_entry.E THEN
			zyl_bandfaenger.st_ctrl.in.b_einfahren := FALSE;
			zyl_bandfaenger.st_ctrl.in.b_ausfahren := FALSE;
			zyl_bandklemmen.st_ctrl.in.b_einfahren := FALSE;
			zyl_bandklemmen.st_ctrl.in.b_ausfahren := FALSE;
			(* Alle Nocken aktivieren, damit die Zylinder wieder winkelgesteuert werden *)
			subr_ST_Bandeinzugsnocken_ein();

			zyl_bandfaenger.fb.b_no_gesteuert_im_norm_betrieb := FALSE;
			zyl_bandklemmen.fb.b_no_gesteuert_im_norm_betrieb := FALSE;
		END_IF

		(*-----------------------Weiterschaltbedingungen----------------------------*)
		fb_state_entry.i16_next_step := 370;

(*=======================================================*)
	370: (* Band neu eingefädelt: Fahre Einfädelhübe und starte dann wieder Bestückzyklus *)
		IF fb_state_entry.E THEN
			fb_virt_master_axis.mc_richtung_modulo :=  MC_Positive_Direction  ;
			(* Beim automatischen Bandwechsel braucht man wengiger Einfädelhübe bis bestückt werden kann*)
			IF b_automatischer_bandwechsel = TRUE THEN
				fb_virt_master_axis.st_position.r_soll := (gst_datensatz.st_wkz.i16_anzahl_einfaedel_auto_pins * 360.0) + gst_datensatz.st_md.st_md_bestueckachse.lr_startposition;
			ELSE
				fb_virt_master_axis.st_position.r_soll := (gst_datensatz.st_wkz.i16_anzahl_einfaedel_pins * 360.0) + gst_datensatz.st_md.st_md_bestueckachse.lr_startposition;
			END_IF

			st_drive_cmd.enu_cmd := MOVE_MODULO;
			bm_an_visu_hinten :=  visu_hinten.in.texte.txt_bm_einfaedeln[2];(*Anstanzhübe werden aktuell gefahren.*)
		END_IF

		(*-----------------------Weiterschaltbedingungen----------------------------*)
		IF st_drive_cmd.enu_cmd = NO_COMMAND THEN
			subr_ST_Bandeinzugsnocken_ein();
			bm_an_visu_hinten := '';
			fb_state_entry.i16_next_step := 380;
		END_IF

(*=======================================================*)
	380:(* Band Scannen*)
		IF 	fb_state_entry.E THEN
			bm_an_visu_hinten :=  visu_hinten.in.texte.txt_bm_einfaedeln[3];(*Band scannen*)
		END_IF

		IF 	(gst_barcode_daten.b_band_links_ok AND gst_barcode_daten.b_band_ID_links_ok AND zyl_bandeinzuege_verschieben.st_ctrl.out.b_ausgefahren)OR
			(gst_barcode_daten.b_band_rechts_ok AND gst_barcode_daten.b_band_ID_rechts_ok AND zyl_bandeinzuege_verschieben.st_ctrl.out.b_eingefahren)
			THEN
				IF	ST_TippTasten.b_einfaedeln_aktiv THEN
					IF 	gst_datensatz.st_md.b_auto_Bandwechsel THEN
						fb_state_entry.i16_next_step := BEREIT;
					ELSE
						sm_fehler_nach_bandwechsel := TRUE;
						(* Dieser Fehler soll kommen, damit Bediener Chargennummer des Bandes ins LTS einträgt, Wunsch von Sebastian Hechenrieder 27.11.17 *)
						fb_state_entry.i16_next_step := FEHLER;(*BEREIT*)
					END_IF
				ELSE
					IF i16_merker_last_state = 150 THEN
						(* Bandende während Bestückablauf *)
						fb_state_entry.i16_next_step := 390;
					ELSE
						(* Bandende aus Step BEREIT *)
						fb_state_entry.i16_next_step := i16_merker_last_state;
					END_IF
				END_IF
		END_IF

		IF fb_state_entry.X THEN
			ST_TippTasten.b_einfaedeln_aktiv:=FALSE;
			b_merker_bandende_links := FALSE;
			b_merker_bandende_rechts := FALSE;
			bm_an_visu_hinten := '';
		END_IF

(*=======================================================*)
	390:	(* Fahre vorgegebene Anzahl von Bestückhüben *)
		IF fb_state_entry.E THEN
			fb_virt_master_axis.st_position.r_soll := (DINT_TO_LREAL(gst_datensatz.st_bestueckprogramm.i32_anzahl - i16_bestueckposzaehler)) * 360.0 + gst_datensatz.st_md.st_md_bestueckachse.lr_startposition;
			st_drive_cmd.enu_cmd := MOVE_MODULO;	(* Achtung beim MODULO-Befehl: fährt nur bis 360° *)
			fb_virt_master_axis.mc_richtung_modulo := MC_Positive_Direction ;
		END_IF

		(*-----------------------Weiterschaltbedingungen----------------------------*)
		IF fb_r_trig_bestueckhubzaehler.Q THEN
			(* Zählt die gesetzten Pins während des gesamten Bestückvorganges *)
			i16_bestueckposzaehler := i16_bestueckposzaehler + 1;
			(* Sobald ein Pin gesetzt wurde wird in den regulären Ablauf mit Camming gesprungen *)
			fb_state_entry.i16_next_step := 150;
		END_IF

(*=======================================================*)
	420:	(* Meldung und warte auf Bediener *)
		IF fb_state_entry.E THEN
			ST_TippTasten.b_einfaedeln_aktiv := TRUE;
			subr_ST_Bandeinzugsnocken_aus();
			bandeinzug_kontroller.st_ctrl.in.b_freigabe := FALSE;           (* GLS überwachung ausschalten*)

			bm_beide_Bandklemmen_oeffnen := TRUE;

			bm_an_visu_hinten :=  visu_hinten.in.texte.txt_bm_einfaedeln[11];(*beide Bandklemmen öffnen -> Taste TIPPEN.*)

			gi16_anzahl_Teile_autostop_bandwechsel := 0;
		END_IF

		IF ST_TippTasten.r_trig_tippen_einfaedeln.Q THEN

			bm_beide_Bandklemmen_oeffnen := FALSE;
			bm_an_visu_hinten := '';
			fb_ton_wz.PT := t#200ms;
			fb_ton_wz.IN := TRUE;

			(* Gib beide Bänder frei *)
			zyl_bandfaenger_li.st_ctrl.in.b_einfahren := TRUE;
			zyl_bandfaenger_li.st_ctrl.in.b_ausfahren := FALSE;
			zyl_bandklemmen_li.st_ctrl.in.b_einfahren := TRUE;
			zyl_bandklemmen_li.st_ctrl.in.b_ausfahren := FALSE;

			zyl_bandfaenger_re.st_ctrl.in.b_einfahren := TRUE;
			zyl_bandfaenger_re.st_ctrl.in.b_ausfahren := FALSE;
			zyl_bandklemmen_re.st_ctrl.in.b_einfahren := TRUE;
			zyl_bandklemmen_re.st_ctrl.in.b_ausfahren := FALSE;
		END_IF

		(*-----------------------Weiterschaltbedingungen----------------------------*)
		IF fb_ton_wz.Q THEN
			IF 	zyl_bandfaenger_li.st_ctrl.out.b_eingefahren AND
				zyl_bandklemmen_li.st_ctrl.out.b_eingefahren AND
				zyl_bandfaenger_re.st_ctrl.out.b_eingefahren AND
				zyl_bandklemmen_re.st_ctrl.out.b_eingefahren
				THEN
					zyl_bandfaenger_li.st_ctrl.in.b_einfahren := FALSE;
					zyl_bandklemmen_li.st_ctrl.in.b_einfahren := FALSE;
					zyl_bandfaenger_re.st_ctrl.in.b_einfahren := FALSE;
					zyl_bandklemmen_re.st_ctrl.in.b_einfahren := FALSE;
					IF i16_merker_last_state = 150 THEN
						fb_state_entry.i16_next_step := 425;
					ELSE
						fb_state_entry.i16_next_step := 440;
					END_IF
			END_IF
		END_IF

(*=======================================================*)
	425: (* Bestückachse mit Bandeinzug steht. Virtuelle Masterachse nochmals eine Umdrehung fahren ohne zu Bestücken, damit Z und Y noch eine Position weiter fahren *)
		IF fb_state_entry.E THEN
			st_drive_cmd.enu_cmd := MOVE_MODULO;
			fb_virt_master_axis.mc_richtung_modulo := MC_Positive_Direction  ;
(**)			fb_virt_master_axis.st_position.r_soll := 360 + gst_datensatz.st_md.st_md_bestueckachse.lr_startposition;
			fb_berechnung_override_achse.lr_skalierung_slave_achse1 := fb_berechnung_override_achse.lr_skalierung_slave_achse2 := 1;
			bandeinzug_kontroller.st_ctrl.in.b_freigabe := FALSE;
		END_IF

		IF fb_r_trig_bestueckhubzaehler.Q THEN
			(* Positionsüberwachung Achsen *)
			subr_ST_PosUW_Z_Achse();

			(* Den Bestückposzähler hier nicht erhöhen, weil auch kein Pin gesetzt wird *)
			i16_bestueckposzaehler := i16_bestueckposzaehler + 1;
		END_IF

		(* Warte auf OT-Nocken für Skalierungsfreigabe *)
		IF fb_f_trig_ot.Q THEN
			(* Skalierung der Kurvenscheibe *)
			subr_ST_Cam_Bestueckachse();
		END_IF

		(* Warte auf Nocken für die Skalierungsfreigabe *)
		IF fb_r_trig_skalierungsnocken.Q THEN
			(* Skalierung der Kurvenscheibe *)
			subr_ST_Cam_Z_Achse();
		END_IF

		(*-----------------------Weiterschaltbedingungen----------------------------*)
		(* Bestückachse auf Startposition *)
		IF	virtuelle_master_achse.Status.NotMoving  AND virtuelle_master_achse.Status.InTargetPosition AND
			st_drive_cmd.enu_cmd = NO_COMMAND AND
			st_drive_cmd_z_achse.enu_cmd = NO_COMMAND
			THEN
				fb_state_entry.i16_next_step := 430;
		END_IF

(*=======================================================*)
	430:	(* Z-Achse muss entkoppelt werden, damit sie bei den Einfädelhüben nicht mitfahren *)
		IF fb_state_entry.E THEN
			st_drive_cmd_z_achse.enu_cmd := CAM_OUT_SLAVE;
		END_IF

		(*-----------------------Weiterschaltbedingungen----------------------------*)
		IF st_drive_cmd_z_achse.enu_cmd = NO_COMMAND THEN
			fb_state_entry.i16_next_step := 440;
		END_IF

(*=======================================================*)
	440:	(* Meldung und warte auf Bediener *)
		IF fb_state_entry.E THEN
			bm_bandende_beide_einzuege_erreicht := FALSE;
			bm_einzug_links_band_entnehmen := TRUE;
			bm_einzug_rechts_band_entnehmen := TRUE;
			bm_an_visu_hinten :=  visu_hinten.in.texte.txt_bm_einfaedeln[4];(*Band an beiden Einzügen entnehmen -> Taste TIPPEN.*)
		END_IF

		(*-----------------------Weiterschaltbedingungen----------------------------*)
		(* Bei Tastendruck darf sich kein Band im entsprechenden Einzug befinden *)
		IF	 ST_TippTasten.r_trig_tippen_einfaedeln.Q AND
			NOT e_ls_bandende_li AND NOT e_ls_bandende_re THEN
			fb_state_entry.i16_next_step := 450;
		END_IF

(*=======================================================*)
	450:	(* Gearin Bestückachse  *)
		IF fb_state_entry.E THEN
			fb_axis_bestueckachse.r_getriebefaktor := axis_bestueckachse.st_config.r_getriebefaktor;
			st_drive_cmd_bestueckachse.enu_cmd := GEAR_IN_SLAVE;
		END_IF

		(*-----------------------Weiterschaltbedingungen----------------------------*)
		IF st_drive_cmd_bestueckachse.enu_cmd = NO_COMMAND THEN
			fb_state_entry.i16_next_step := 455;
		END_IF

(*=======================================================*)
	455:	(* Fahre auf UT *)
		IF fb_state_entry.E THEN
			bm_einzug_links_band_entnehmen := FALSE;
			bm_einzug_rechts_band_entnehmen := FALSE;
			bm_an_visu_hinten := '';

			fb_virt_master_axis.mc_richtung_modulo :=  MC_Positive_Direction  ;
			fb_virt_master_axis.st_position.r_soll := gst_datensatz.st_wkz.lr_einfaedelposition;
			st_drive_cmd.enu_cmd := MOVE_MODULO;
		END_IF

		(*-----------------------Weiterschaltbedingungen----------------------------*)
		IF st_drive_cmd.enu_cmd = NO_COMMAND THEN
			fb_state_entry.i16_next_step := 460;
		END_IF

(*=======================================================*)
	460:	(* Meldung und warte auf Bediener *)
		IF fb_state_entry.E THEN
			bm_einzug_links_band_auf_anschlag := TRUE;
			bm_einzug_rechts_band_auf_anschlag := TRUE;
			bm_an_visu_hinten :=  visu_hinten.in.texte.txt_bm_einfaedeln[7];(*Band an beiden Einzügen auf Anschlag in WKZ -> Taste TIPPEN.*)
		END_IF

		IF ST_TippTasten.r_trig_tippen_einfaedeln.Q THEN
			bm_einzug_links_band_auf_anschlag := FALSE;
			bm_einzug_rechts_band_auf_anschlag := FALSE;
			bm_an_visu_hinten := '';
			fb_ton_wz.PT := t#200ms;
			fb_ton_wz.IN := TRUE;

			(* Zylinder ausfahren *)
			(* Klemme das Linke und Rechte Band *)
			zyl_bandfaenger_li.st_ctrl.in.b_einfahren := TRUE;
			zyl_bandfaenger_li.st_ctrl.in.b_ausfahren := FALSE;
			zyl_bandklemmen_li.st_ctrl.in.b_einfahren := FALSE;
			zyl_bandklemmen_li.st_ctrl.in.b_ausfahren := TRUE;

			zyl_bandfaenger_re.st_ctrl.in.b_einfahren := TRUE;
			zyl_bandfaenger_re.st_ctrl.in.b_ausfahren := FALSE;
			zyl_bandklemmen_re.st_ctrl.in.b_einfahren := FALSE;
			zyl_bandklemmen_re.st_ctrl.in.b_ausfahren := TRUE;
		END_IF

		(*-----------------------Weiterschaltbedingungen----------------------------*)
		IF fb_ton_wz.Q THEN
			IF 	zyl_bandfaenger_li.st_ctrl.out.b_eingefahren AND
				zyl_bandklemmen_li.st_ctrl.out.b_ausgefahren AND
				zyl_bandfaenger_re.st_ctrl.out.b_eingefahren AND
				zyl_bandklemmen_re.st_ctrl.out.b_ausgefahren
				THEN
					zyl_bandfaenger_li.st_ctrl.in.b_einfahren := FALSE;
					zyl_bandklemmen_li.st_ctrl.in.b_ausfahren := FALSE;
					zyl_bandfaenger_re.st_ctrl.in.b_einfahren := FALSE;
					zyl_bandklemmen_re.st_ctrl.in.b_ausfahren := FALSE;
					fb_state_entry.i16_next_step := 470;
					fb_ton_wz.IN := FALSE;
			END_IF
		END_IF

(*=======================================================*)
	470:	(* Warte kurz auf Zylinder *)
		IF fb_state_entry.E THEN
 			fb_ton_wz.PT := t#1s;
			fb_ton_wz.IN := TRUE;
		END_IF

		(*-----------------------Weiterschaltbedingungen----------------------------*)
		IF fb_ton_wz.Q THEN
			fb_ton_wz.IN := FALSE;
			fb_state_entry.i16_next_step := 475;
		END_IF

(*=======================================================*)
	475:	(* Fahre auf OT - beide Bänder sind geklemmt *)
		IF fb_state_entry.E THEN
			fb_virt_master_axis.mc_richtung_modulo :=  MC_Positive_Direction  ;
			fb_virt_master_axis.st_position.r_soll := gst_datensatz.st_md.st_md_bestueckachse.lr_startposition;
			st_drive_cmd.enu_cmd := MOVE_MODULO;
			bm_an_visu_hinten :=  visu_hinten.in.texte.txt_bm_einfaedeln[1];(*Werkzeug fährt auf OT.*)
		END_IF

		(*-----------------------Weiterschaltbedingungen----------------------------*)
		IF st_drive_cmd.enu_cmd = NO_COMMAND THEN
			fb_state_entry.i16_next_step := 480;
		END_IF

(*=======================================================*)
	480:	(* Entsprechende Zylinder wieder den Nocken überlassen *)

		(* Links -> Nockenfahrt / Rechts -> Nockenfahrt *)
		zyl_bandfaenger_li.st_ctrl.in.b_einfahren := FALSE;
		zyl_bandfaenger_li.st_ctrl.in.b_ausfahren := FALSE;
		zyl_bandklemmen_li.st_ctrl.in.b_einfahren := FALSE;
		zyl_bandklemmen_li.st_ctrl.in.b_ausfahren := FALSE;

		zyl_bandfaenger_re.st_ctrl.in.b_einfahren := FALSE;
		zyl_bandfaenger_re.st_ctrl.in.b_ausfahren := FALSE;
		zyl_bandklemmen_re.st_ctrl.in.b_einfahren := FALSE;
		zyl_bandklemmen_re.st_ctrl.in.b_ausfahren := FALSE;

		(* Alle Nocken aktivieren, damit die Zylinder wieder winkelgesteuert werden *)
		subr_ST_Bandeinzugsnocken_ein();

		zyl_bandfaenger_li.fb.b_no_gesteuert_im_norm_betrieb := FALSE;
		zyl_bandklemmen_li.fb.b_no_gesteuert_im_norm_betrieb := FALSE;
		zyl_bandfaenger_re.fb.b_no_gesteuert_im_norm_betrieb := FALSE;
		zyl_bandklemmen_re.fb.b_no_gesteuert_im_norm_betrieb := FALSE;

		fb_state_entry.i16_next_step := 490;

(*=======================================================*)
	490: (* Band neu eingefädelt: Fahre Einfädelhübe und starte dann wieder Bestückzyklus *)
		IF fb_state_entry.E THEN
			fb_virt_master_axis.mc_richtung_modulo :=  MC_Positive_Direction  ;
			fb_virt_master_axis.st_position.r_soll := (INT_TO_LREAL(gst_datensatz.st_wkz.i16_anzahl_einfaedel_pins)) * 360.0 + gst_datensatz.st_md.st_md_bestueckachse.lr_startposition;
			st_drive_cmd.enu_cmd := MOVE_MODULO;
			bm_an_visu_hinten :=  visu_hinten.in.texte.txt_bm_einfaedeln[2];(*Anstanzhübe werden aktuell gefahren.*)
		END_IF

		(*-----------------------Weiterschaltbedingungen----------------------------*)
		IF st_drive_cmd.enu_cmd = NO_COMMAND THEN

			(* Alle Nocken aktivieren, damit die Zylinder wieder winkelgesteuert werden *)
			subr_ST_Bandeinzugsnocken_ein();

			bm_an_visu_hinten := '';
			bm_an_visu_hinten := '';

			fb_state_entry.i16_next_step := 500;
		END_IF

(*=======================================================*)
	500:(* Band Scannen*)
		IF 	fb_state_entry.E THEN
			bm_an_visu_hinten :=  visu_hinten.in.texte.txt_bm_einfaedeln[3];(*Band scannen*)
		END_IF

		(*-----------------------Weiterschaltbedingungen----------------------------*)
		IF gst_barcode_daten.b_band_ok THEN
			IF	ST_TippTasten.b_einfaedeln_aktiv  THEN
				fb_state_entry.i16_next_step := BEREIT;
			ELSE
				IF i16_merker_last_state = 150 THEN
					(* Bandende während Bestückablauf *)
					fb_state_entry.i16_next_step := 510;
				ELSE
					(* Bandende aus Step BEREIT oder Step 110 *)
					fb_state_entry.i16_next_step := i16_merker_last_state;
				END_IF
			END_IF
		END_IF

		IF fb_state_entry.X THEN
			ST_TippTasten.b_einfaedeln_aktiv:=FALSE;
			b_merker_bandende_links := FALSE;
			b_merker_bandende_rechts := FALSE;
			bm_an_visu_hinten := '';
		END_IF

(*=======================================================*)
	510:	(* Fahre vorgegebene Anzahl von Bestückhüben *)
		IF fb_state_entry.E THEN
			fb_virt_master_axis.st_position.r_soll := (DINT_TO_LREAL(gst_datensatz.st_bestueckprogramm.i32_anzahl - i16_bestueckposzaehler)) * 360.0 + gst_datensatz.st_md.st_md_bestueckachse.lr_startposition;
			st_drive_cmd.enu_cmd := MOVE_MODULO;	(* Achtung beim MODULO-Befehl: fährt nur bis 360° *)
			fb_virt_master_axis.mc_richtung_modulo :=MC_Positive_Direction ;
		END_IF

		(*-----------------------Weiterschaltbedingungen----------------------------*)
		fb_state_entry.i16_next_step := 150;

(*=======================================================*)
	640:	(* Cam_in_Slave*)
		IF fb_state_entry.E THEN
			ST_TippTasten.b_einfaedeln_aktiv := TRUE;
			b_einfaedeln_aktiv_servo := TRUE;
			bandeinzug_kontroller.st_ctrl.in.b_freigabe := FALSE;           (* GLS überwachung ausschalten*)
			i16_bestueckachse_cam_table_id := 5;
			fb_axis_bestueckachse.mc_activation_mode_camin:= MC_CAMACTIVATION_ATMASTERCAMPOS;
			fb_axis_bestueckachse.lr_activation_position_camin := gst_datensatz.st_md.st_md_bestueckachse.lr_startposition;
			st_drive_cmd_bestueckachse.enu_cmd := CAM_IN_SLAVE;
			i16_bestueckachse_cam_table_id_alt := i16_bestueckachse_cam_table_id;
		END_IF

		(*-----------------------Weiterschaltbedingungen----------------------------*)
		IF st_drive_cmd_bestueckachse.enu_cmd = NO_COMMAND AND NOT fb_state_entry.E THEN
			fb_state_entry.i16_next_step := 645;
		END_IF

(*=======================================================*)
	645:	(* Starte automatischen Bandwechsel bzw. manueller Wechsel bis Band heraus gezogen wurde *)
		(* Die Bremse des Servobandeinzugs wird im Bandwechselablauf angesteuert *)
		IF fb_state_entry.E THEN
			bandwechsel_kontroller.st_ctrl.in.b_start := TRUE;
			fb_ton_wz.pt := t#300ms;
			fb_ton_wz.IN := TRUE;
			gi16_anzahl_Teile_autostop_bandwechsel := 0;
		END_IF

		(*-----------------------Weiterschaltbedingungen----------------------------*)
		IF bandwechsel_kontroller.st_ctrl.out.b_fertig AND NOT fb_state_entry.E AND fb_ton_wz.Q THEN
		(*Bandwechsel ist vollzogen und die Seite wurde getauscht *)
			bandwechsel_kontroller.st_ctrl.in.b_start := FALSE;
			bm_bandende_einzug_links_erreicht := FALSE;
			bm_bandende_einzug_rechts_erreicht := FALSE;
			fb_ton_wz.IN := FALSE;
			fb_state_entry.i16_next_step := 650;
		(*Es ist kein Band im anderen Einzug. Gleiche Seite wird wieder verwendet *)
		ELSIF bandwechsel_kontroller.st_ctrl.out.b_fertig_2 AND NOT fb_state_entry.E AND fb_ton_wz.Q THEN
			bandwechsel_kontroller.st_ctrl.in.b_start := FALSE;
			bm_bandende_einzug_links_erreicht := FALSE;
			bm_bandende_einzug_rechts_erreicht := FALSE;
			fb_ton_wz.IN := FALSE;
			fb_state_entry.i16_next_step := 700;
		END_IF

(*=======================================================*)
	650:	(* Gearin Bestückachse  *)
		IF fb_state_entry.E THEN
			fb_axis_bestueckachse.r_getriebefaktor := axis_bestueckachse.st_config.r_getriebefaktor;
			st_drive_cmd_bestueckachse.enu_cmd := GEAR_IN_SLAVE;
		END_IF

		(*-----------------------Weiterschaltbedingungen----------------------------*)
		IF st_drive_cmd_bestueckachse.enu_cmd = NO_COMMAND AND NOT fb_state_entry.E THEN
			fb_state_entry.i16_next_step := 655;
		END_IF

(*=======================================================*)
	655:	(* Fahre auf UT *)
		IF fb_state_entry.E THEN
			fb_virt_master_axis.mc_richtung_modulo :=  MC_Positive_Direction  ;
			fb_virt_master_axis.st_position.r_soll := gst_datensatz.st_wkz.lr_einfaedelposition;
			st_drive_cmd.enu_cmd := MOVE_MODULO;
		END_IF

		(*-----------------------Weiterschaltbedingungen----------------------------*)
		IF st_drive_cmd.enu_cmd = NO_COMMAND THEN
			fb_state_entry.i16_next_step := 660;
		END_IF

(*=======================================================*)
	660:	(* Starte Einfädelprozedur Servobandeinzug *)
		IF fb_state_entry.E THEN
			axis_bandeinzug_achse.st_ctrl.in.b_start := TRUE;
			axis_bandeinzug_achse.st_ctrl.in.b_einfaedeln_servo := TRUE;
		END_IF

		(*-----------------------Weiterschaltbedingungen----------------------------*)
		IF axis_bandeinzug_achse.st_ctrl.out.b_fertig AND NOT fb_state_entry.E THEN
			axis_bandeinzug_achse.st_ctrl.in.b_start := FALSE;
			axis_bandeinzug_achse.st_ctrl.in.b_einfaedeln_servo := FALSE;
			fb_state_entry.i16_next_step := 665;
		END_IF

(*=======================================================*)
	665:	(* Bremse an Servobandeinzug wieder fest. *)
		IF fb_state_entry.E THEN
			axis_bandeinzug_achse.st_ctrl.in.b_bremse_zu := TRUE;
		END_IF

		(*-----------------------Weiterschaltbedingungen----------------------------*)
		IF axis_bandeinzug_achse.st_ctrl.out.b_bremse_geschlossen AND NOT fb_state_entry.E THEN
			axis_bandeinzug_achse.st_ctrl.in.b_bremse_zu := FALSE;
			fb_state_entry.i16_next_step := 670; (* Überspringe schreiben *)
		END_IF

(*=======================================================*)
	670:	(* Fahre auf OT - Band ist fest *)
		IF fb_state_entry.E THEN
			fb_virt_master_axis.mc_richtung_modulo :=  MC_Positive_Direction  ;
			fb_virt_master_axis.st_position.r_soll := gst_datensatz.st_md.st_md_bestueckachse.lr_startposition;
			st_drive_cmd.enu_cmd := MOVE_MODULO;
			bm_an_visu_hinten :=  visu_hinten.in.texte.txt_bm_einfaedeln[1];(*Werkzeug fährt auf OT.*)
		END_IF

		(*-----------------------Weiterschaltbedingungen----------------------------*)
		IF st_drive_cmd.enu_cmd = NO_COMMAND THEN
			fb_state_entry.i16_next_step := 675;
		END_IF

(*=======================================================*)
	675:	(* Band neu eingefädelt: Fahre Einfädelhübe und starte dann wieder Bestückzyklus *)
		IF fb_state_entry.E THEN
			st_drive_cmd.enu_cmd := MOVE_MODULO;
			fb_virt_master_axis.mc_richtung_modulo :=  MC_Positive_Direction  ;
			fb_virt_master_axis.st_position.r_soll := gst_datensatz.st_wkz.i16_anzahl_einfaedel_pins * 360.0 + gst_datensatz.st_md.st_md_bestueckachse.lr_startposition;
			i16_einfaedelzaehler := 0;
			bm_an_visu_hinten :=  visu_hinten.in.texte.txt_bm_einfaedeln[2];(*Anstanzhübe werden aktuell gefahren.*)
		END_IF

		(* Warte auf Nocken für die Skalierungsfreigabe *)
		IF fb_r_trig_skalierungsnocken.Q THEN
			fb_axis_b_achse.st_camscaling_data.SlaveScaling := F_Servobandeinzug_Strecke_zu_Grad( strecke := gst_datensatz.st_band.r_raster);
			i16_einfaedelzaehler := i16_einfaedelzaehler + 1;

			IF b_achse.Status.CamScalingPending THEN
				st_sm.b_skalierung_noch_aktiv := TRUE;
				fb_state_entry.i16_next_step := FEHLER;
			ELSE
				IF b_achse.NcToPlc.CoupleState = 0 THEN
					st_drive_cmd_b_achse.enu_cmd := CAM_IN_SLAVE;
				ELSE
					st_drive_cmd_b_achse.enu_cmd := CAM_SCALEING_SLAVE;
				END_IF
			END_IF
		END_IF

		(*-----------------------Weiterschaltbedingungen----------------------------*)
		IF st_drive_cmd.enu_cmd = NO_COMMAND AND st_drive_cmd_b_achse.enu_cmd = NO_COMMAND THEN;
			ST_TippTasten.b_einfaedeln_aktiv := FALSE;
			b_einfaedeln_aktiv_servo := FALSE;
			bm_an_visu_hinten := '';
			IF i16_merker_last_state = 100 THEN
				fb_state_entry.i16_next_step := BEREIT;
			ELSIF i16_merker_last_state = 150 THEN
				fb_state_entry.i16_next_step := 680;
			ELSE
				sm_fehler_nach_bandwechsel := TRUE;
				(* Dieser Fehler soll kommen, damit Bediener Chargennummer des Bandes ins LTS einträgt, Wunsch von Sebastian Hechenrieder 27.11.17 *)
				fb_state_entry.i16_next_step := FEHLER;(*BEREIT*)
			END_IF
		END_IF

(*=======================================================*)
	680:	(* Fahre vorgegebene Anzahl von Bestückhüben *)
		IF fb_state_entry.E THEN
			fb_virt_master_axis.st_position.r_soll := (DINT_TO_LREAL(gst_datensatz.st_bestueckprogramm.i32_anzahl - i16_bestueckposzaehler)) * 360.0 + gst_datensatz.st_md.st_md_bestueckachse.lr_startposition;
			st_drive_cmd.enu_cmd := MOVE_MODULO;	(* Achtung beim MODULO-Befehl: fährt nur bis 360° *)
			fb_virt_master_axis.mc_richtung_modulo :=MC_Positive_Direction ;
		END_IF

		(* Warte auf Nocken für die Skalierungsfreigabe *)
		IF fb_r_trig_skalierungsnocken.Q THEN
			subr_ST_Cam_B_Achse();
		END_IF

		(*-----------------------Weiterschaltbedingungen----------------------------*)
		IF fb_r_trig_bestueckhubzaehler.Q THEN
			(* Zählt die gesetzten Pins während des gesamten Bestückvorganges *)
			i16_bestueckposzaehler := i16_bestueckposzaehler + 1;
			(* Sobald ein Pin gesetzt wurde, wird in den regulären Ablauf mit Camming gesprungen *)
			fb_state_entry.i16_next_step := 150;
		END_IF

(*---------------------------------------------------------------------------------------------------------------------------------------------------------------------------------------------------*)
(*===========================Anstanzen 1700 mit Servobandeinzug============================*)
	700:	(* Bandende im linken oder rechten Einzug ohne Bandwechsel ->Meldung und warte auf Bediener *)
		IF fb_state_entry.E THEN
			bm_bandende_einzug_links_erreicht := FALSE;
			bm_bandende_einzug_rechts_erreicht := FALSE;
			IF b_merker_bandende_links THEN
				bm_einzug_links_band_entnehmen := TRUE;
			ELSIF b_merker_bandende_rechts THEN
				bm_einzug_rechts_band_entnehmen := TRUE;
			END_IF
			bm_an_visu_hinten :=  visu_hinten.in.texte.txt_bm_einfaedeln[0];(*Band am Einzug entnehmen -> Taste TIPPEN.*)
		END_IF

		(*-----------------------Weiterschaltbedingungen----------------------------*)
		IF ST_TippTasten.r_trig_tippen_einfaedeln.Q THEN
			(* Bei Tastendruck darf sich kein Band im Einzug befinden *)
			IF b_merker_bandende_links THEN
				IF NOT e_ls_bandende_li THEN
					fb_state_entry.i16_next_step := 710;
				END_IF
			ELSIF b_merker_bandende_rechts THEN
				IF NOT e_ls_bandende_re THEN
					fb_state_entry.i16_next_step := 710;
				END_IF
			END_IF
		END_IF

(*=======================================================*)
	710:	(* Gearin Bestückachse  *)
		IF fb_state_entry.E THEN
			fb_axis_bestueckachse.r_getriebefaktor := axis_bestueckachse.st_config.r_getriebefaktor;
			st_drive_cmd_bestueckachse.enu_cmd := GEAR_IN_SLAVE;
		END_IF

		(*-----------------------Weiterschaltbedingungen----------------------------*)
		IF st_drive_cmd_bestueckachse.enu_cmd = NO_COMMAND AND NOT fb_state_entry.E THEN
			fb_state_entry.i16_next_step := 720;
		END_IF

(*=======================================================*)
	720:	(* Fahre auf UT *)
		IF fb_state_entry.E THEN
			bm_einzug_links_band_entnehmen := FALSE;
			bm_einzug_rechts_band_entnehmen := FALSE;
			bm_an_visu_hinten := '';

			fb_virt_master_axis.mc_richtung_modulo :=  MC_Positive_Direction  ;
			fb_virt_master_axis.st_position.r_soll := gst_datensatz.st_wkz.lr_einfaedelposition;
			st_drive_cmd.enu_cmd := MOVE_MODULO;
		END_IF

		(*-----------------------Weiterschaltbedingungen----------------------------*)
		IF st_drive_cmd.enu_cmd = NO_COMMAND THEN
			fb_state_entry.i16_next_step := 725;
		END_IF

(*=======================================================*)
	725:	(* Fahre Igelrad auf Position*)
		IF fb_state_entry.E THEN
			axis_bandeinzug_achse.st_ctrl.in.b_startpos := TRUE;
			fb_ton_wz.PT := t#100ms;
			fb_ton_wz.IN := TRUE;
		END_IF

		(*-----------------------Weiterschaltbedingungen----------------------------*)
		IF axis_bandeinzug_achse.st_ctrl.out.b_servo_auf_einfaedelpos AND fb_ton_wz.Q THEN
			axis_bandeinzug_achse.st_ctrl.in.b_startpos := FALSE;
			fb_state_entry.i16_next_step := 730;
		END_IF

		IF fb_state_entry.X THEN
			fb_ton_wz.IN := FALSE;
		END_IF

(*=======================================================*)
	730:	(* Meldung Band in Igelrad einführen *)
		IF fb_state_entry.E THEN
			IF b_merker_bandende_links THEN
				bm_einzug_links_band_bis_gls := TRUE;
			ELSIF b_merker_bandende_rechts THEN
				bm_einzug_rechts_band_bis_gls := TRUE;
			END_IF
			bm_an_visu_hinten :=  visu_hinten.in.texte.txt_bm_einfaedeln[10];(*Band bis zum Igelrad einschieben -> Taste Servo manuell fahren *)
		END_IF

		(*-----------------------Weiterschaltbedingungen----------------------------*)
		fb_state_entry.i16_next_step := 735;

(*=======================================================*)
	735:	(* Starte Einfädelprozedur Servobandeinzug *)
		IF fb_state_entry.E THEN
			axis_bandeinzug_achse.st_ctrl.in.b_start := TRUE;
		END_IF

		(*-----------------------Weiterschaltbedingungen----------------------------*)
		IF axis_bandeinzug_achse.st_ctrl.out.b_fertig AND NOT fb_state_entry.E THEN
			axis_bandeinzug_achse.st_ctrl.in.b_start := FALSE;
			fb_state_entry.i16_next_step := 740;
		END_IF

(*=======================================================*)
	740:	(* Bremse an Servobandeinzug wieder fest. *)
		IF fb_state_entry.E THEN
			axis_bandeinzug_achse.st_ctrl.in.b_bremse_zu := TRUE;
			bm_einzug_rechts_band_bis_gls := FALSE;
			bm_einzug_links_band_bis_gls := FALSE;
			bm_an_visu_hinten := '';
		END_IF

		(*-----------------------Weiterschaltbedingungen----------------------------*)
		IF axis_bandeinzug_achse.st_ctrl.out.b_bremse_geschlossen AND NOT fb_state_entry.E THEN
			axis_bandeinzug_achse.st_ctrl.in.b_bremse_zu := FALSE;
			fb_state_entry.i16_next_step := 750;
		END_IF

(*=======================================================*)
	750:	(* Fahre auf OT - Band ist fest *)
		IF fb_state_entry.E THEN
			fb_virt_master_axis.mc_richtung_modulo :=  MC_Positive_Direction  ;
			fb_virt_master_axis.st_position.r_soll := gst_datensatz.st_md.st_md_bestueckachse.lr_startposition;
			st_drive_cmd.enu_cmd := MOVE_MODULO;
			bm_an_visu_hinten :=  visu_hinten.in.texte.txt_bm_einfaedeln[1];(*Werkzeug fährt auf OT.*)
		END_IF

		(*-----------------------Weiterschaltbedingungen----------------------------*)
		IF st_drive_cmd.enu_cmd = NO_COMMAND THEN
			fb_state_entry.i16_next_step := 770;
		END_IF

(*=======================================================*)
	770:	(* Band neu eingefädelt: Fahre Einfädelhübe und starte dann wieder Bestückzyklus *)
		IF fb_state_entry.E THEN
			st_drive_cmd.enu_cmd := MOVE_MODULO;
			fb_virt_master_axis.mc_richtung_modulo :=  MC_Positive_Direction  ;
			fb_virt_master_axis.st_position.r_soll := gst_datensatz.st_wkz.i16_anzahl_einfaedel_pins * 360.0 + gst_datensatz.st_md.st_md_bestueckachse.lr_startposition;
			i16_einfaedelzaehler := 0;
			bm_an_visu_hinten :=  visu_hinten.in.texte.txt_bm_einfaedeln[2];(*Anstanzhübe werden aktuell gefahren.*)
		END_IF

		(* Warte auf Nocken für die Skalierungsfreigabe *)
		IF fb_r_trig_skalierungsnocken.Q THEN
			IF (i16_einfaedelzaehler = 0) THEN
				fb_axis_b_achse.st_camscaling_data.SlaveScaling := F_Servobandeinzug_Strecke_zu_Grad( strecke := gst_datensatz.st_band.r_raster + gst_datensatz.st_band.lr_offset_erster_hub_wkz_mm);
			ELSE
				fb_axis_b_achse.st_camscaling_data.SlaveScaling := F_Servobandeinzug_Strecke_zu_Grad( strecke := gst_datensatz.st_band.r_raster);
			END_IF
			i16_einfaedelzaehler := i16_einfaedelzaehler + 1;

			IF b_achse.Status.CamScalingPending THEN
				st_sm.b_skalierung_noch_aktiv := TRUE;
				fb_state_entry.i16_next_step := FEHLER;
			ELSE
				IF b_achse.NcToPlc.CoupleState = 0 THEN
					st_drive_cmd_b_achse.enu_cmd := CAM_IN_SLAVE;
				ELSE
					st_drive_cmd_b_achse.enu_cmd := CAM_SCALEING_SLAVE;
				END_IF
			END_IF
		END_IF

		(*-----------------------Weiterschaltbedingungen----------------------------*)
		IF st_drive_cmd.enu_cmd = NO_COMMAND THEN
			bm_an_visu_hinten := '';
			b_einfaedeln_aktiv_servo := FALSE;
			fb_state_entry.i16_next_step := 780;
		END_IF

(*=======================================================*)
	780:	(* Band Scannen*)
		IF 	fb_state_entry.E THEN
			bm_an_visu_hinten :=  visu_hinten.in.texte.txt_bm_einfaedeln[3];(*Band scannen*)
		END_IF

		IF 	(gst_barcode_daten.b_band_links_ok AND gst_barcode_daten.b_band_ID_links_ok AND zyl_bandeinzuege_verschieben.st_ctrl.out.b_ausgefahren)OR
			(gst_barcode_daten.b_band_rechts_ok AND gst_barcode_daten.b_band_ID_rechts_ok AND zyl_bandeinzuege_verschieben.st_ctrl.out.b_eingefahren)
			THEN
				IF	ST_TippTasten.b_einfaedeln_aktiv THEN
					fb_state_entry.i16_next_step := BEREIT;
				ELSE
					IF i16_merker_last_state = 150 THEN
						(* Bandende während Bestückablauf *)
						fb_state_entry.i16_next_step := 790;
					ELSE
						(* Bandende aus Step BEREIT *)
						fb_state_entry.i16_next_step := BEREIT;
					END_IF
				END_IF
		END_IF

		IF fb_state_entry.X THEN
			ST_TippTasten.b_einfaedeln_aktiv:=FALSE;
			b_merker_bandende_links := FALSE;
			b_merker_bandende_rechts := FALSE;
			bm_an_visu_hinten := '';
		END_IF

(*=======================================================*)
	790:	(* Fahre vorgegebene Anzahl von Bestückhüben *)
		IF fb_state_entry.E THEN
			fb_virt_master_axis.st_position.r_soll := ((gst_datensatz.st_bestueckprogramm.i32_anzahl - i16_bestueckposzaehler) * 360.0) + gst_datensatz.st_md.st_md_bestueckachse.lr_startposition;
			st_drive_cmd.enu_cmd := MOVE_MODULO;	(* Achtung beim MODULO-Befehl: fährt nur bis 360° *)
			fb_virt_master_axis.mc_richtung_modulo :=MC_Positive_Direction ;
			ST_TippTasten.b_einfaedeln_aktiv := FALSE;
		END_IF

		(* Warte auf Nocken für die Skalierungsfreigabe *)
		IF fb_r_trig_skalierungsnocken.Q THEN
			subr_ST_Cam_B_Achse();
		END_IF

		(*-----------------------Weiterschaltbedingungen----------------------------*)
		IF fb_r_trig_bestueckhubzaehler.Q THEN
			(* Zählt die gesetzten Pins während des gesamten Bestückvorganges *)
			i16_bestueckposzaehler := i16_bestueckposzaehler + 1;
			(* Sobald ein Pin gesetzt wurde wird in den regulären Ablauf mit Camming gesprungen *)
			fb_state_entry.i16_next_step := 150;
		END_IF

(*---------------------------------------------------------------------------------------------------------------------------------------------------------------------------------------------------*)
(*===========================Rasterfolie============================*)
	800:	(* Fahre nur einen Hub zum Rasterfolien setzen *)
		IF fb_state_entry.E THEN
			fb_virt_master_axis.mc_richtung_modulo :=  MC_Positive_Direction  ;
			fb_virt_master_axis.st_position.r_soll := 360 + gst_datensatz.st_md.st_md_bestueckachse.lr_startposition;
			st_drive_cmd.enu_cmd := MOVE_MODULO;
		END_IF

		(* Rasterfolieneinzug lüften
		Dies wird nur gemacht, wenn die Nocken ungleich 0 sind und Anfangs- und Endnocke aunterschiedlich sind 
		Zwischen den Nocken wird die Rasterfolie vom Werkzeug gehalten *)
		IF gst_datensatz.st_wkz.nockenschaltwerk_bestueckachse.arr_nocken[NO_RASTERFOLIE_LUEFTEN].r_cam_begin <> 0 AND
			gst_datensatz.st_wkz.nockenschaltwerk_bestueckachse.arr_nocken[NO_RASTERFOLIE_LUEFTEN].r_cam_begin <> gst_datensatz.st_wkz.nockenschaltwerk_bestueckachse.arr_nocken[NO_RASTERFOLIE_LUEFTEN].r_cam_end THEN
			IF st_visu.i32_position_ist > gst_datensatz.st_wkz.nockenschaltwerk_bestueckachse.arr_nocken[NO_RASTERFOLIE_LUEFTEN].r_cam_begin AND
				st_visu.i32_position_ist < (gst_datensatz.st_wkz.nockenschaltwerk_bestueckachse.arr_nocken[NO_RASTERFOLIE_LUEFTEN].r_cam_begin + 5) THEN
				zyl_rafo_klemmen.st_ctrl.in.b_einfahren := TRUE;
			ELSE
				zyl_rafo_klemmen.st_ctrl.in.b_einfahren := FALSE;
			END_IF

			IF st_visu.i32_position_ist > gst_datensatz.st_wkz.nockenschaltwerk_bestueckachse.arr_nocken[NO_RASTERFOLIE_LUEFTEN].r_cam_end AND
				st_visu.i32_position_ist < (gst_datensatz.st_wkz.nockenschaltwerk_bestueckachse.arr_nocken[NO_RASTERFOLIE_LUEFTEN].r_cam_end + 5) THEN
				zyl_rafo_faenger.st_ctrl.in.b_ausfahren := TRUE;
			ELSE
				zyl_rafo_faenger.st_ctrl.in.b_ausfahren := FALSE;
			END_IF
		END_IF

		(*-----------------------Weiterschaltbedingungen----------------------------*)
		IF st_drive_cmd.enu_cmd = NO_COMMAND THEN
			fb_state_entry.i16_next_step := BEREIT;
		END_IF

(*===========================Rasterfolie Einfädelvorgang============================*)
	810:	(* Fänger einfahren, damit das Band drunter geschoben werden kann *)
		IF fb_state_entry.E THEN
			ST_TippTasten.b_einfaedeln_aktiv:=TRUE;
			zyl_rafo_faenger.st_ctrl.in.b_einfahren := TRUE;
		END_IF

		(*-----------------------Weiterschaltbedingungen----------------------------*)
		IF zyl_rafo_faenger.st_ctrl.out.b_eingefahren THEN
			zyl_rafo_faenger.st_ctrl.in.b_einfahren := FALSE;
			bm_an_visu_hinten :=  visu_hinten.in.texte.txt_bm_einfaedeln[0];(*Band am Einzug entnehmen -> Taste TIPPEN.*)
			IF ST_TippTasten.r_trig_tippen_einfaedeln.Q  THEN
				fb_state_entry.i16_next_step := 820;
			END_IF
		END_IF

(*=======================================================*)
	820:	(* Meldung fahre Werkzeug auf UT *)
		IF fb_state_entry.E THEN
			bm_an_visu_hinten := '';
			fb_virt_master_axis.mc_richtung_modulo :=  MC_Positive_Direction  ;
			fb_virt_master_axis.st_position.r_soll := gst_datensatz.st_wkz.lr_einfaedelposition;
			st_drive_cmd.enu_cmd := MOVE_MODULO;
		END_IF

		(*-----------------------Weiterschaltbedingungen----------------------------*)
		IF st_drive_cmd.enu_cmd = NO_COMMAND THEN
			fb_state_entry.i16_next_step := 830;
		END_IF

(*=======================================================*)
	830:	(* Rasterfolie von Hand einschieben und bestätigen *)

		IF fb_state_entry.E THEN
			bm_einzug_links_band_auf_anschlag := TRUE;
			bm_an_visu_hinten :=  visu_hinten.in.texte.txt_bm_einfaedeln[8];(*Band an Einzug links auf Anschlag in WKZ -> Taste TIPPEN.*)
		END_IF

		IF ST_TippTasten.r_trig_tippen_einfaedeln.Q  THEN
			bm_einzug_links_band_auf_anschlag := FALSE;
			bm_an_visu_hinten := '';

			(* Fange das Band *)
			zyl_rafo_faenger.st_ctrl.in.b_einfahren := FALSE;
			zyl_rafo_faenger.st_ctrl.in.b_ausfahren := TRUE;
		END_IF

		(*-----------------------Weiterschaltbedingungen----------------------------*)
		IF zyl_rafo_faenger.st_ctrl.out.b_ausgefahren THEN
			zyl_rafo_faenger.st_ctrl.in.b_ausfahren := FALSE;
			fb_state_entry.i16_next_step := 840;
		END_IF

(*=======================================================*)
	840:	(* Fahre auf OT - Band ist fest *)
		IF fb_state_entry.E THEN
			fb_virt_master_axis.mc_richtung_modulo :=  MC_Positive_Direction  ;
			fb_virt_master_axis.st_position.r_soll := gst_datensatz.st_md.st_md_bestueckachse.lr_startposition;
			st_drive_cmd.enu_cmd := MOVE_MODULO;
			bm_an_visu_hinten :=  visu_hinten.in.texte.txt_bm_einfaedeln[1];(*Werkzeug fährt auf OT.*)
		END_IF

		(*-----------------------Weiterschaltbedingungen----------------------------*)
		IF st_drive_cmd.enu_cmd = NO_COMMAND THEN
			bm_an_visu_hinten := '';
			ST_TippTasten.b_einfaedeln_aktiv := FALSE;
			fb_state_entry.i16_next_step := BEREIT;
		END_IF

(*---------------------------------------------------------------------------------------------------------------------------------------------------------------------------------------------------*)
(*===========================Werkzeug Ausbauposition============================*)
	900:	(* Fahre zur Ausbauposition des Werkzeugs *)
		IF fb_state_entry.E THEN
			fb_virt_master_axis.mc_richtung_modulo :=  MC_Positive_Direction  ;
			fb_virt_master_axis.st_position.r_soll := gst_datensatz.st_wkz.lr_ausbauposition;
			st_drive_cmd.enu_cmd := MOVE_MODULO;
		END_IF

		(*-----------------------Weiterschaltbedingungen----------------------------*)
		IF st_drive_cmd.enu_cmd = NO_COMMAND THEN
			fb_state_entry.i16_next_step := 905;
		END_IF

(*=======================================================*)
	905: (*Warten bis keine ander Produktions Meldung ansteht *)
		IF	TestAndSet(ST_Message_Produktion.LockFlag) THEN
			ST_Message_Produktion.ClearMessageLines();
			fb_state_entry.i16_next_step := 910;
		END_IF

(*=======================================================*)
	910:  (*Produktions Meldung*)
		Visu.MeldungProduktion.Color_R := 255;
		Visu.MeldungProduktion.Color_G := 0;
		Visu.MeldungProduktion.Color_B := 0;
		IF visu.s_akt_sprache = 'de' THEN
			Visu.MeldungProduktion.Name:='Werkzeug kann ausgebaut werden. Weiter mit OK';
		ELSIF visu.s_akt_sprache = 'en' THEN
			Visu.MeldungProduktion.Name:='Tool can now be removed. Confirm with OK';
		ELSIF visu.s_akt_sprache = 'cz' THEN
			Visu.MeldungProduktion.Name:='Nastroj muze byt vyjmut. Pokracovat pres OK';
		END_IF
		Visu.MeldungProduktion.ShowMessage := TRUE;
		Visu.MeldungProduktion.Button1.sichtbar:=TRUE;	(*OK*)
		Visu.MeldungProduktion.Button1.Text:='Ok';
		fb_state_entry.i16_next_step := 915;

(*=======================================================*)
	915:  (*Warte auf OK*)
		IF Visu.MeldungProduktion.Button1.tasten THEN
			fb_state_entry.i16_next_step:=FEHLER;
		END_IF

(*=======================================================*)
	FEHLER:
		IF fb_state_entry.E THEN
			st_ctrl_out.b_fehler := TRUE;
			fb_ton_quitt.IN := FALSE;

		END_IF

		(*-----------------------Weiterschaltbedingungen----------------------------*)
		IF st_ctrl_in.b_quitt AND NOT fb_state_entry.E THEN
			st_ctrl_out.b_fehler := FALSE;
			st_drive_cmd.enu_cmd := RESET;
			st_drive_cmd_bestueckachse.enu_cmd := RESET;
			st_drive_cmd_z_achse.enu_cmd := RESET;
			st_drive_cmd_y_achse.enu_cmd := RESET;
			st_drive_cmd_b_achse.enu_cmd := RESET;
			fb_ton_quitt.IN := TRUE;

		END_IF

		IF st_ctrl_in.b_stop AND NOT virtuelle_master_achse.Status.HasBeenStopped THEN
			st_drive_cmd.enu_cmd := STOP_AXIS;
		END_IF

		IF st_ctrl_in.b_halt AND virtuelle_master_achse.Status.Moving THEN
			st_drive_cmd.enu_cmd := HALT_AXIS;
			st_geschwindigkeiten.lr_verzoegerung := lr_decceleration_nothalt;
		END_IF

		IF fb_ton_quitt.Q THEN
			fb_ton_quitt.IN := FALSE;
			fb_state_entry.i16_next_step := INIT;
		END_IF

(*=======================================================*)
	STOP:
		IF fb_state_entry.E THEN
			st_drive_cmd.enu_cmd := STOP_AXIS;
		END_IF

		(*-----------------------Weiterschaltbedingungen----------------------------*)
		IF st_drive_cmd.enu_cmd = NO_COMMAND AND virtuelle_master_achse.Status.NotMoving THEN
			fb_state_entry.i16_next_step := STILLSTAND;
		END_IF

(*=======================================================*)
	STILLSTAND:
		IF fb_state_entry.E THEN
			st_drive_cmd.enu_cmd := POWER_DISABLE;
			fb_ton_quitt.IN := FALSE;

		END_IF

		(*-----------------------Weiterschaltbedingungen----------------------------*)
		IF st_ctrl_in.b_quitt AND NOT fb_state_entry.E THEN
			fb_ton_quitt.IN := TRUE;
		END_IF

		IF fb_ton_quitt.Q THEN
			fb_ton_quitt.IN := FALSE;
			fb_state_entry.i16_next_step := INIT;
		END_IF

(*=======================================================*)
	HALT:
		IF fb_state_entry.E THEN
			st_drive_cmd.enu_cmd := HALT_AXIS;
			st_geschwindigkeiten.lr_verzoegerung := lr_decceleration_nothalt;
			fb_ton_quitt.IN := FALSE;
		END_IF

		(*-----------------------Weiterschaltbedingungen----------------------------*)
		IF st_ctrl_in.b_quitt AND NOT fb_state_entry.E THEN
			fb_ton_quitt.IN := TRUE;
		END_IF

		IF fb_ton_quitt.Q THEN
			fb_ton_quitt.IN := FALSE;
			fb_state_entry.i16_next_step := INIT;
		END_IF
END_CASE

fb_state_entry(
	i16_next_step:= , 
	i16_pos:= 2,
	s_debugtext:= ,
	E=> ,
	X=> ,
	i16_step=> ,
	i16_last_step=> );

IF st_config_achse.b_config_fertig THEN
	(* Fehlermeldungen und Betriebsmeldungen ab dem Startindex in die globalen Meldungsarrays schreiben *)
	garr_stoermeldungen[st_config_achse.i16_meld_startindex + 0] := st_sm.b_achse_nicht_bb;
	garr_stoermeldungen[st_config_achse.i16_meld_startindex + 1] := st_sm.b_achse_nicht_referenziert;
	garr_stoermeldungen[st_config_achse.i16_meld_startindex + 2] := st_sm.b_keine_verfahrfreigabe;
	garr_stoermeldungen[st_config_achse.i16_meld_startindex + 3] := st_sm.b_achse_nicht_auf_startpos;
	garr_stoermeldungen[st_config_achse.i16_meld_startindex + 4] := st_sm.b_ende_skalierungs_nocke;
	garr_stoermeldungen[st_config_achse.i16_meld_startindex + 5] := st_sm.b_ende_camming_nocke;
	garr_stoermeldungen[st_config_achse.i16_meld_startindex + 6] := st_sm.b_skalierung_noch_aktiv;
	garr_stoermeldungen[st_config_achse.i16_meld_startindex + 7] := FALSE;
	garr_stoermeldungen[st_config_achse.i16_meld_startindex + 8] := FALSE;
	garr_stoermeldungen[st_config_achse.i16_meld_startindex + 9] := sm_fehler_raster_oder_zaehne;
	garr_stoermeldungen[st_config_achse.i16_meld_startindex + 10] := FALSE;
	garr_stoermeldungen[st_config_achse.i16_meld_startindex + 11] := FALSE;
	garr_stoermeldungen[st_config_achse.i16_meld_startindex + 12] := sm_fehler_achse_lueften;
	garr_stoermeldungen[st_config_achse.i16_meld_startindex + 13] := sm_keine_busverbindung;
	garr_stoermeldungen[st_config_achse.i16_meld_startindex + 14] := sm_fehler_bestueckanzahl;
	garr_stoermeldungen[st_config_achse.i16_meld_startindex + 15] := sm_fehler_nach_bandwechsel;
	garr_stoermeldungen[st_config_achse.i16_meld_startindex + 16] := st_drive_cmd.meldungen.sm_write_soe_parameter;
	garr_stoermeldungen[st_config_achse.i16_meld_startindex + 17] := st_drive_cmd.meldungen.sm_read_soe_parameter;
	garr_stoermeldungen[st_config_achse.i16_meld_startindex + 18] := st_drive_cmd.meldungen.sm_write_nc_parameter;
	garr_stoermeldungen[st_config_achse.i16_meld_startindex + 19] := st_drive_cmd.meldungen.sm_read_nc_parameter;
	garr_stoermeldungen[st_config_achse.i16_meld_startindex + 20] := st_drive_cmd.meldungen.sm_power_enable;
	garr_stoermeldungen[st_config_achse.i16_meld_startindex + 21] := st_drive_cmd.meldungen.sm_power_disable;
	garr_stoermeldungen[st_config_achse.i16_meld_startindex + 22] := st_drive_cmd.meldungen.sm_reset;
	garr_stoermeldungen[st_config_achse.i16_meld_startindex + 23] := st_drive_cmd.meldungen.sm_home;
	garr_stoermeldungen[st_config_achse.i16_meld_startindex + 24] := st_drive_cmd.meldungen.sm_setposition;
	garr_stoermeldungen[st_config_achse.i16_meld_startindex + 25] := st_drive_cmd.meldungen.sm_jog_vorwaerts;
	garr_stoermeldungen[st_config_achse.i16_meld_startindex + 26] := st_drive_cmd.meldungen.sm_jog_rueckwaerts;
	garr_stoermeldungen[st_config_achse.i16_meld_startindex + 27] := st_drive_cmd.meldungen.sm_move_absolute;
	garr_stoermeldungen[st_config_achse.i16_meld_startindex + 28] := st_drive_cmd.meldungen.sm_move_relative;
	garr_stoermeldungen[st_config_achse.i16_meld_startindex + 29] := st_drive_cmd.meldungen.sm_move_velocity;
	garr_stoermeldungen[st_config_achse.i16_meld_startindex + 30] := st_drive_cmd.meldungen.sm_move_modulo;
	garr_stoermeldungen[st_config_achse.i16_meld_startindex + 31] := st_drive_cmd.meldungen.sm_stop_axis;
	garr_stoermeldungen[st_config_achse.i16_meld_startindex + 32] := st_drive_cmd.meldungen.sm_halt_axis;
	garr_stoermeldungen[st_config_achse.i16_meld_startindex + 33] := st_drive_cmd.meldungen.sm_motion_command_timeout;
	garr_stoermeldungen[st_config_achse.i16_meld_startindex + 34] := st_sm.b_achsfehler;
	garr_stoermeldungen[st_config_achse.i16_meld_startindex + 35] := st_sm.b_devicefehler;
	garr_stoermeldungen[st_config_achse.i16_meld_startindex + 36] := st_drive_cmd.meldungen.sm_limit_positiv_erreicht;
	garr_stoermeldungen[st_config_achse.i16_meld_startindex + 37] := st_drive_cmd.meldungen.sm_limit_negativ_erreicht;
	garr_stoermeldungen[st_config_achse.i16_meld_startindex + 38] := st_drive_cmd.meldungen.sm_ec_coe_sdo_write_ex;
	garr_stoermeldungen[st_config_achse.i16_meld_startindex + 39] := st_drive_cmd.meldungen.sm_ec_coe_sdo_read_ex;
	garr_stoermeldungen[st_config_achse.i16_meld_startindex + 40] := st_drive_cmd_z_achse.meldungen.sm_gear_in_slave;
	garr_stoermeldungen[st_config_achse.i16_meld_startindex + 41] := st_drive_cmd_z_achse.meldungen.sm_gear_out_slave;
	garr_stoermeldungen[st_config_achse.i16_meld_startindex + 42] := st_drive_cmd_z_achse.meldungen.sm_cam_in_slave;
	garr_stoermeldungen[st_config_achse.i16_meld_startindex + 43] := st_drive_cmd_z_achse.meldungen.sm_cam_out_slave;
	garr_stoermeldungen[st_config_achse.i16_meld_startindex + 44] := st_drive_cmd_z_achse.meldungen.sm_cam_scaleing_slave;
	garr_stoermeldungen[st_config_achse.i16_meld_startindex + 45] := st_drive_cmd_z_achse.meldungen.sm_camgear_command_timeout;
	garr_stoermeldungen[st_config_achse.i16_meld_startindex + 46] := st_drive_cmd_z_achse.meldungen.sm_read_motion_funktion_point;
	garr_stoermeldungen[st_config_achse.i16_meld_startindex + 47] := st_drive_cmd_z_achse.meldungen.sm_write_motion_funktion_point;
	garr_stoermeldungen[st_config_achse.i16_meld_startindex + 48] := st_drive_cmd_z_achse.meldungen.sm_read_camtable_slave_dynamics;
	garr_stoermeldungen[st_config_achse.i16_meld_startindex + 49] := st_drive_cmd_z_achse.meldungen.sm_read_camtable_charakteristik;
	garr_stoermeldungen[st_config_achse.i16_meld_startindex + 50] := st_drive_cmd_y_achse.meldungen.sm_gear_in_slave;
	garr_stoermeldungen[st_config_achse.i16_meld_startindex + 51] := st_drive_cmd_y_achse.meldungen.sm_gear_out_slave;
	garr_stoermeldungen[st_config_achse.i16_meld_startindex + 52] := st_drive_cmd_y_achse.meldungen.sm_cam_in_slave;
	garr_stoermeldungen[st_config_achse.i16_meld_startindex + 53] := st_drive_cmd_y_achse.meldungen.sm_cam_out_slave;
	garr_stoermeldungen[st_config_achse.i16_meld_startindex + 54] := st_drive_cmd_y_achse.meldungen.sm_cam_scaleing_slave;
	garr_stoermeldungen[st_config_achse.i16_meld_startindex + 55] := st_drive_cmd_y_achse.meldungen.sm_camgear_command_timeout;
	garr_stoermeldungen[st_config_achse.i16_meld_startindex + 56] := st_drive_cmd_y_achse.meldungen.sm_read_motion_funktion_point;
	garr_stoermeldungen[st_config_achse.i16_meld_startindex + 57] := st_drive_cmd_y_achse.meldungen.sm_write_motion_funktion_point;
	garr_stoermeldungen[st_config_achse.i16_meld_startindex + 58] := st_drive_cmd_y_achse.meldungen.sm_read_camtable_slave_dynamics;
	garr_stoermeldungen[st_config_achse.i16_meld_startindex + 59] := st_drive_cmd_y_achse.meldungen.sm_read_camtable_charakteristik;
	garr_stoermeldungen[st_config_achse.i16_meld_startindex + 60] := st_drive_cmd_b_achse.meldungen.sm_gear_in_slave;
	garr_stoermeldungen[st_config_achse.i16_meld_startindex + 61] := st_drive_cmd_b_achse.meldungen.sm_gear_out_slave;
	garr_stoermeldungen[st_config_achse.i16_meld_startindex + 62] := st_drive_cmd_b_achse.meldungen.sm_cam_in_slave;
	garr_stoermeldungen[st_config_achse.i16_meld_startindex + 63] := st_drive_cmd_b_achse.meldungen.sm_cam_out_slave;
	garr_stoermeldungen[st_config_achse.i16_meld_startindex + 64] := st_drive_cmd_b_achse.meldungen.sm_cam_scaleing_slave;
	garr_stoermeldungen[st_config_achse.i16_meld_startindex + 65] := st_drive_cmd_b_achse.meldungen.sm_camgear_command_timeout;
	garr_stoermeldungen[st_config_achse.i16_meld_startindex + 66] := st_drive_cmd_b_achse.meldungen.sm_read_motion_funktion_point;
	garr_stoermeldungen[st_config_achse.i16_meld_startindex + 67] := st_drive_cmd_b_achse.meldungen.sm_write_motion_funktion_point;
	garr_stoermeldungen[st_config_achse.i16_meld_startindex + 68] := st_drive_cmd_b_achse.meldungen.sm_read_camtable_slave_dynamics;
	garr_stoermeldungen[st_config_achse.i16_meld_startindex + 69] := st_drive_cmd_b_achse.meldungen.sm_read_camtable_charakteristik;
	garr_stoermeldungen[st_config_achse.i16_meld_startindex + 70] :=  sm_fehler_positionierung_z;
	garr_stoermeldungen[st_config_achse.i16_meld_startindex + 71] :=  sm_fehler_positionierung_y;
	garr_stoermeldungen[st_config_achse.i16_meld_startindex + 72] :=  sm_fehler_bestueckschieberanzahl;
	garr_stoermeldungen[st_config_achse.i16_meld_startindex + 73] :=  sm_fehler_bestueckposition_z;
	garr_stoermeldungen[st_config_achse.i16_meld_startindex + 74] :=  sm_fehler_bestueckposition_y;
	garr_stoermeldungen[st_config_achse.i16_meld_startindex + 75] :=  sm_fehler_positionierung_bestueckachse;
	garr_stoermeldungen[st_config_achse.i16_meld_startindex + 76] :=  st_drive_cmd_bestueckachse.meldungen.sm_gear_in_slave;
	garr_stoermeldungen[st_config_achse.i16_meld_startindex + 77] :=  st_drive_cmd_bestueckachse.meldungen.sm_gear_out_slave;
	garr_stoermeldungen[st_config_achse.i16_meld_startindex + 78] :=  st_drive_cmd_bestueckachse.meldungen.sm_cam_in_slave;
	garr_stoermeldungen[st_config_achse.i16_meld_startindex + 79] :=  st_drive_cmd_bestueckachse.meldungen.sm_cam_out_slave;
	garr_stoermeldungen[st_config_achse.i16_meld_startindex + 80] :=  st_drive_cmd_bestueckachse.meldungen.sm_camgear_command_timeout;
	garr_stoermeldungen[st_config_achse.i16_meld_startindex + 81] :=  st_drive_cmd_bestueckachse.meldungen.sm_read_motion_funktion_point;
	garr_stoermeldungen[st_config_achse.i16_meld_startindex + 82] :=  st_drive_cmd_bestueckachse.meldungen.sm_write_motion_funktion_point;
	garr_stoermeldungen[st_config_achse.i16_meld_startindex + 83] :=  st_drive_cmd_bestueckachse.meldungen.sm_read_camtable_slave_dynamics;
	garr_stoermeldungen[st_config_achse.i16_meld_startindex + 84] :=  st_drive_cmd_bestueckachse.meldungen.sm_read_camtable_charakteristik;
	garr_stoermeldungen[st_config_achse.i16_meld_startindex + 85] :=  FALSE;
	garr_stoermeldungen[st_config_achse.i16_meld_startindex + 86] :=  FALSE;
	garr_stoermeldungen[st_config_achse.i16_meld_startindex + 87] :=  FALSE;
	garr_stoermeldungen[st_config_achse.i16_meld_startindex + 88] :=  FALSE;
	garr_stoermeldungen[st_config_achse.i16_meld_startindex + 89] :=  FALSE;
	garr_stoermeldungen[st_config_achse.i16_meld_startindex + 90] :=  FALSE;
	garr_stoermeldungen[st_config_achse.i16_meld_startindex + 91] :=  FALSE;
	garr_stoermeldungen[st_config_achse.i16_meld_startindex + 92] :=  FALSE;
	garr_stoermeldungen[st_config_achse.i16_meld_startindex + 93] :=  FALSE;
	garr_stoermeldungen[st_config_achse.i16_meld_startindex + 94] :=  FALSE;
	garr_stoermeldungen[st_config_achse.i16_meld_startindex + 95] :=  FALSE;
	garr_stoermeldungen[st_config_achse.i16_meld_startindex + 96] :=  FALSE;
	garr_stoermeldungen[st_config_achse.i16_meld_startindex + 97] :=  FALSE;
	garr_stoermeldungen[st_config_achse.i16_meld_startindex + 98] :=  FALSE;
	garr_stoermeldungen[st_config_achse.i16_meld_startindex + 99] :=  FALSE;
	
	garr_betriebsmeldungen[st_config_achse.i16_meld_startindex + 0] := bm_bandende_einzug_links_erreicht;
	garr_betriebsmeldungen[st_config_achse.i16_meld_startindex + 1] := bm_einzug_links_band_entnehmen;
	garr_betriebsmeldungen[st_config_achse.i16_meld_startindex + 2] := bm_einzug_links_band_auf_anschlag;
	garr_betriebsmeldungen[st_config_achse.i16_meld_startindex + 3] := FALSE;
	garr_betriebsmeldungen[st_config_achse.i16_meld_startindex + 4] := FALSE;
	garr_betriebsmeldungen[st_config_achse.i16_meld_startindex + 5] := FALSE;
	garr_betriebsmeldungen[st_config_achse.i16_meld_startindex + 6] := FALSE;
	garr_betriebsmeldungen[st_config_achse.i16_meld_startindex + 7] := FALSE;
	garr_betriebsmeldungen[st_config_achse.i16_meld_startindex + 8] := FALSE;
	garr_betriebsmeldungen[st_config_achse.i16_meld_startindex + 9] := FALSE;
	garr_betriebsmeldungen[st_config_achse.i16_meld_startindex + 10] := bm_bandende_einzug_rechts_erreicht;
	garr_betriebsmeldungen[st_config_achse.i16_meld_startindex + 11] := bm_einzug_rechts_band_entnehmen;
	garr_betriebsmeldungen[st_config_achse.i16_meld_startindex + 12] := bm_einzug_rechts_band_auf_anschlag;
	garr_betriebsmeldungen[st_config_achse.i16_meld_startindex + 13] := FALSE;
	garr_betriebsmeldungen[st_config_achse.i16_meld_startindex + 14] := FALSE;
	garr_betriebsmeldungen[st_config_achse.i16_meld_startindex + 15] := FALSE;
	garr_betriebsmeldungen[st_config_achse.i16_meld_startindex + 16] := FALSE;
	garr_betriebsmeldungen[st_config_achse.i16_meld_startindex + 17] := FALSE;
	garr_betriebsmeldungen[st_config_achse.i16_meld_startindex + 18] := FALSE;
	garr_betriebsmeldungen[st_config_achse.i16_meld_startindex + 19] := FALSE;
	garr_betriebsmeldungen[st_config_achse.i16_meld_startindex + 20] := bm_bandende_beide_einzuege_erreicht;
	garr_betriebsmeldungen[st_config_achse.i16_meld_startindex + 21] := bm_override_kleiner_stufe9;
	garr_betriebsmeldungen[st_config_achse.i16_meld_startindex + 22] := bm_md_offset_z_pos_0_zu_hoch;
	garr_betriebsmeldungen[st_config_achse.i16_meld_startindex + 23] := bm_md_offset_y_pos_0_zu_hoch;
	garr_betriebsmeldungen[st_config_achse.i16_meld_startindex + 24] := FALSE;
	garr_betriebsmeldungen[st_config_achse.i16_meld_startindex + 25] := FALSE;
	garr_betriebsmeldungen[st_config_achse.i16_meld_startindex + 26] := FALSE;
	garr_betriebsmeldungen[st_config_achse.i16_meld_startindex + 27] := FALSE;
	garr_betriebsmeldungen[st_config_achse.i16_meld_startindex + 28] := FALSE;
	garr_betriebsmeldungen[st_config_achse.i16_meld_startindex + 29] := FALSE;
	garr_betriebsmeldungen[st_config_achse.i16_meld_startindex + 30] := FALSE;
	garr_betriebsmeldungen[st_config_achse.i16_meld_startindex + 31] := FALSE;
	garr_betriebsmeldungen[st_config_achse.i16_meld_startindex + 32] := FALSE;
	garr_betriebsmeldungen[st_config_achse.i16_meld_startindex + 33] := FALSE;
	garr_betriebsmeldungen[st_config_achse.i16_meld_startindex + 34] := FALSE;
	garr_betriebsmeldungen[st_config_achse.i16_meld_startindex + 35] := FALSE;
	garr_betriebsmeldungen[st_config_achse.i16_meld_startindex + 36] := FALSE;
	garr_betriebsmeldungen[st_config_achse.i16_meld_startindex + 37] := FALSE;
	garr_betriebsmeldungen[st_config_achse.i16_meld_startindex + 38] := FALSE;
	garr_betriebsmeldungen[st_config_achse.i16_meld_startindex + 39] := FALSE;
	garr_betriebsmeldungen[st_config_achse.i16_meld_startindex + 40] := FALSE;
	garr_betriebsmeldungen[st_config_achse.i16_meld_startindex + 41] := FALSE;
	garr_betriebsmeldungen[st_config_achse.i16_meld_startindex + 42] := FALSE;
	garr_betriebsmeldungen[st_config_achse.i16_meld_startindex + 43] := FALSE;
	garr_betriebsmeldungen[st_config_achse.i16_meld_startindex + 44] := FALSE;
	garr_betriebsmeldungen[st_config_achse.i16_meld_startindex + 45] := FALSE;
	garr_betriebsmeldungen[st_config_achse.i16_meld_startindex + 46] := FALSE;
	garr_betriebsmeldungen[st_config_achse.i16_meld_startindex + 47] := FALSE;
	garr_betriebsmeldungen[st_config_achse.i16_meld_startindex + 48] := FALSE;
	garr_betriebsmeldungen[st_config_achse.i16_meld_startindex + 49] := FALSE;
	garr_betriebsmeldungen[st_config_achse.i16_meld_startindex + 50] := FALSE;
	garr_betriebsmeldungen[st_config_achse.i16_meld_startindex + 51] := FALSE;
	garr_betriebsmeldungen[st_config_achse.i16_meld_startindex + 52] := FALSE;
	garr_betriebsmeldungen[st_config_achse.i16_meld_startindex + 53] := FALSE;
	garr_betriebsmeldungen[st_config_achse.i16_meld_startindex + 54] := FALSE;
	garr_betriebsmeldungen[st_config_achse.i16_meld_startindex + 55] := FALSE;
	garr_betriebsmeldungen[st_config_achse.i16_meld_startindex + 56] := FALSE;
	garr_betriebsmeldungen[st_config_achse.i16_meld_startindex + 57] := FALSE;
	garr_betriebsmeldungen[st_config_achse.i16_meld_startindex + 58] := FALSE;
	garr_betriebsmeldungen[st_config_achse.i16_meld_startindex + 59] := FALSE;
	garr_betriebsmeldungen[st_config_achse.i16_meld_startindex + 60] := FALSE;
	garr_betriebsmeldungen[st_config_achse.i16_meld_startindex + 61] := FALSE;
	garr_betriebsmeldungen[st_config_achse.i16_meld_startindex + 62] := FALSE;
	garr_betriebsmeldungen[st_config_achse.i16_meld_startindex + 63] := FALSE;
	garr_betriebsmeldungen[st_config_achse.i16_meld_startindex + 64] := FALSE;
	garr_betriebsmeldungen[st_config_achse.i16_meld_startindex + 65] := FALSE;
	garr_betriebsmeldungen[st_config_achse.i16_meld_startindex + 66] := FALSE;
	garr_betriebsmeldungen[st_config_achse.i16_meld_startindex + 67] := FALSE;
	garr_betriebsmeldungen[st_config_achse.i16_meld_startindex + 68] := FALSE;
	garr_betriebsmeldungen[st_config_achse.i16_meld_startindex + 69] := FALSE;
	garr_betriebsmeldungen[st_config_achse.i16_meld_startindex + 70] :=  FALSE;
	garr_betriebsmeldungen[st_config_achse.i16_meld_startindex + 71] :=  FALSE;
	garr_betriebsmeldungen[st_config_achse.i16_meld_startindex + 72] :=  FALSE;
	garr_betriebsmeldungen[st_config_achse.i16_meld_startindex + 73] :=  FALSE;
	garr_betriebsmeldungen[st_config_achse.i16_meld_startindex + 74] :=  FALSE;
	garr_betriebsmeldungen[st_config_achse.i16_meld_startindex + 75] :=  FALSE;
	garr_betriebsmeldungen[st_config_achse.i16_meld_startindex + 76] :=  FALSE;
	garr_betriebsmeldungen[st_config_achse.i16_meld_startindex + 77] :=  FALSE;
	garr_betriebsmeldungen[st_config_achse.i16_meld_startindex + 78] :=  FALSE;
	garr_betriebsmeldungen[st_config_achse.i16_meld_startindex + 79] :=  FALSE;
	garr_betriebsmeldungen[st_config_achse.i16_meld_startindex + 80] :=  FALSE;
	garr_betriebsmeldungen[st_config_achse.i16_meld_startindex + 81] :=  FALSE;
	garr_betriebsmeldungen[st_config_achse.i16_meld_startindex + 82] :=  FALSE;
	garr_betriebsmeldungen[st_config_achse.i16_meld_startindex + 83] :=  FALSE;
	garr_betriebsmeldungen[st_config_achse.i16_meld_startindex + 84] :=  FALSE;
	garr_betriebsmeldungen[st_config_achse.i16_meld_startindex + 85] :=  FALSE;
	garr_betriebsmeldungen[st_config_achse.i16_meld_startindex + 86] :=  FALSE;
	garr_betriebsmeldungen[st_config_achse.i16_meld_startindex + 87] :=  FALSE;
	garr_betriebsmeldungen[st_config_achse.i16_meld_startindex + 88] :=  FALSE;
	garr_betriebsmeldungen[st_config_achse.i16_meld_startindex + 89] :=  FALSE;
	garr_betriebsmeldungen[st_config_achse.i16_meld_startindex + 90] :=  FALSE;
	garr_betriebsmeldungen[st_config_achse.i16_meld_startindex + 91] :=  FALSE;
	garr_betriebsmeldungen[st_config_achse.i16_meld_startindex + 92] :=  FALSE;
	garr_betriebsmeldungen[st_config_achse.i16_meld_startindex + 93] :=  FALSE;
	garr_betriebsmeldungen[st_config_achse.i16_meld_startindex + 94] :=  FALSE;
	garr_betriebsmeldungen[st_config_achse.i16_meld_startindex + 95] :=  FALSE;
	garr_betriebsmeldungen[st_config_achse.i16_meld_startindex + 96] :=  FALSE;
	garr_betriebsmeldungen[st_config_achse.i16_meld_startindex + 97] :=  FALSE;
	garr_betriebsmeldungen[st_config_achse.i16_meld_startindex + 98] :=  FALSE;
	garr_betriebsmeldungen[st_config_achse.i16_meld_startindex + 99] :=  FALSE;
END_IF
END_PROGRAM
ACTION subr_ST_B_Achse:
(* Überwachung, wenn falsche Info aus dem Bestückbild kommt *)
(* Fehler, wenn mehr bestückt werden soll als das WKZ Bestückschieber hat *)
IF gst_datensatz.st_bestueckprogramm.i16_b[i16_bestueckposzaehler] > gst_datensatz.st_wkz.i16_anzahl_bestueckschieber THEN
	sm_fehler_bestueckschieberanzahl := TRUE;
	fb_state_entry.i16_next_step := FEHLER;
END_IF
END_ACTION
ACTION subr_ST_Bandeinzugsnocken_aus:
CASE gst_datensatz.st_wkz.i16_typ_bandeinzug OF
	 STANDARD_2FACH_V2:

		(* Bandeinzug: Standard_2fach_V1 *)
		gst_datensatz.st_wkz.nockenschaltwerk_bestueckachse.arr_nocken[NO_BW_BANDFAENGER_LI_EINFAHREN].b_camvalid := FALSE;
		gst_datensatz.st_wkz.nockenschaltwerk_bestueckachse.arr_nocken[NO_BW_BANDFAENGER_LI_AUSFAHREN].b_camvalid := FALSE;
		gst_datensatz.st_wkz.nockenschaltwerk_bestueckachse.arr_nocken[NO_BW_BANDKLEMMEN_LI_EINFAHREN].b_camvalid := FALSE;
		gst_datensatz.st_wkz.nockenschaltwerk_bestueckachse.arr_nocken[NO_BW_BANDKLEMMEN_LI_AUSFAHREN].b_camvalid := FALSE;
		gst_datensatz.st_wkz.nockenschaltwerk_bestueckachse.arr_nocken[NO_UW_BANDFAENGER_LI_EINFAHREN].b_camvalid := FALSE;
		gst_datensatz.st_wkz.nockenschaltwerk_bestueckachse.arr_nocken[NO_UW_BANDFAENGER_LI_AUSFAHREN].b_camvalid := FALSE;
		gst_datensatz.st_wkz.nockenschaltwerk_bestueckachse.arr_nocken[NO_UW_BANDKLEMMEN_LI_EINFAHREN].b_camvalid := FALSE;
		gst_datensatz.st_wkz.nockenschaltwerk_bestueckachse.arr_nocken[NO_UW_BANDKLEMMEN_LI_AUSFAHREN].b_camvalid := FALSE;
		gst_datensatz.st_wkz.nockenschaltwerk_bestueckachse.arr_nocken[NO_BW_BANDFAENGER_RE_EINFAHREN].b_camvalid := FALSE;
		gst_datensatz.st_wkz.nockenschaltwerk_bestueckachse.arr_nocken[NO_BW_BANDFAENGER_RE_AUSFAHREN].b_camvalid := FALSE;
		gst_datensatz.st_wkz.nockenschaltwerk_bestueckachse.arr_nocken[NO_BW_BANDKLEMMEN_RE_EINFAHREN].b_camvalid := FALSE;
		gst_datensatz.st_wkz.nockenschaltwerk_bestueckachse.arr_nocken[NO_BW_BANDKLEMMEN_RE_AUSFAHREN].b_camvalid := FALSE;
		gst_datensatz.st_wkz.nockenschaltwerk_bestueckachse.arr_nocken[NO_UW_BANDFAENGER_RE_EINFAHREN].b_camvalid := FALSE;
		gst_datensatz.st_wkz.nockenschaltwerk_bestueckachse.arr_nocken[NO_UW_BANDFAENGER_RE_AUSFAHREN].b_camvalid := FALSE;
		gst_datensatz.st_wkz.nockenschaltwerk_bestueckachse.arr_nocken[NO_UW_BANDKLEMMEN_RE_EINFAHREN].b_camvalid := FALSE;
		gst_datensatz.st_wkz.nockenschaltwerk_bestueckachse.arr_nocken[NO_UW_BANDKLEMMEN_RE_AUSFAHREN].b_camvalid := FALSE;
		(* Bandeinzug: Standard_2fach_V2 *)
		gst_datensatz.st_wkz.nockenschaltwerk_bestueckachse.arr_nocken[NO_BW_BANDFAENGER_LI_BAEZV2_EINFAHREN].b_camvalid := FALSE;
		gst_datensatz.st_wkz.nockenschaltwerk_bestueckachse.arr_nocken[NO_BW_BANDFAENGER_LI_BAEZV2_AUSFAHREN].b_camvalid := FALSE;
		gst_datensatz.st_wkz.nockenschaltwerk_bestueckachse.arr_nocken[NO_BW_BANDKLEMMEN_LI_BAEZV2_EINFAHREN].b_camvalid := FALSE;
		gst_datensatz.st_wkz.nockenschaltwerk_bestueckachse.arr_nocken[NO_BW_BANDKLEMMEN_LI_BAEZV2_AUSFAHREN].b_camvalid := FALSE;
		gst_datensatz.st_wkz.nockenschaltwerk_bestueckachse.arr_nocken[NO_BW_BANDFAENGER_RE_BAEZV2_EINFAHREN].b_camvalid := FALSE;
		gst_datensatz.st_wkz.nockenschaltwerk_bestueckachse.arr_nocken[NO_BW_BANDFAENGER_RE_BAEZV2_AUSFAHREN].b_camvalid := FALSE;
		gst_datensatz.st_wkz.nockenschaltwerk_bestueckachse.arr_nocken[NO_BW_BANDKLEMMEN_RE_BAEZV2_EINFAHREN].b_camvalid := FALSE;
		gst_datensatz.st_wkz.nockenschaltwerk_bestueckachse.arr_nocken[NO_BW_BANDKLEMMEN_RE_BAEZV2_AUSFAHREN].b_camvalid := FALSE;

		zyl_bandfaenger_li.fb.b_no_gesteuert_im_norm_betrieb := TRUE;
		zyl_bandklemmen_li.fb.b_no_gesteuert_im_norm_betrieb := TRUE;
		zyl_bandfaenger_re.fb.b_no_gesteuert_im_norm_betrieb := TRUE;
		zyl_bandklemmen_re.fb.b_no_gesteuert_im_norm_betrieb := TRUE;

	BANDWECHSLER_V2:
		(* Klemmbandeinzug ohne Sensoren *)
		gst_datensatz.st_wkz.nockenschaltwerk_bestueckachse.arr_nocken[NO_BW_BANDFAENGER_BAWEV2_EINFAHREN].b_camvalid := FALSE;
		gst_datensatz.st_wkz.nockenschaltwerk_bestueckachse.arr_nocken[NO_BW_BANDFAENGER_BAWEV2_AUSFAHREN].b_camvalid := FALSE;
		gst_datensatz.st_wkz.nockenschaltwerk_bestueckachse.arr_nocken[NO_BW_BANDKLEMMEN_BAWEV2_EINFAHREN].b_camvalid := FALSE;
		gst_datensatz.st_wkz.nockenschaltwerk_bestueckachse.arr_nocken[NO_BW_BANDKLEMMEN_BAWEV2_AUSFAHREN].b_camvalid := FALSE;

